KUKA KRL program: EPS_2_25369_MH4A_A_20251215023758.src

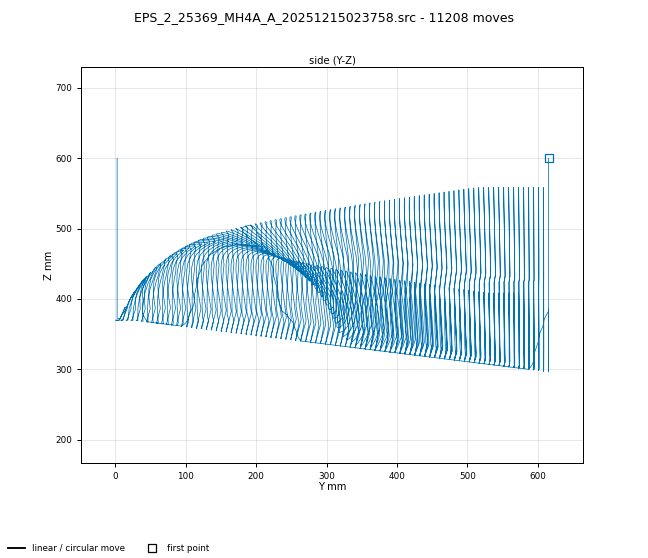
[picture p0: tool path of EPS_2_25369_MH4A_A_20251215023758.src, 11208 of 11210 moves have a stored position in this frame; points joined in program order, loops and branches not executed]
&ACCESS RVP
&REL 4
&COMMENT QRS 19112012
&PARAM EDITMASK = *
DEF PART()
EXT BAS (BAS_COMMAND :IN,REAL :IN )
INT I
BAS (#INITMOV,0 )

;KUKA QRS Post kuka4.cps  Date:22-06-2017 !

File_ID=2957

QRS_PRE_INIT()

;Init var - Until changes are made in qrs_pre_init
Outlet_Square_prg=0
Inlet_1_Square_prg=0
Inlet_2_Square_prg=0
Inlet_3_Square_prg=0
Inlet_4_Square_prg=0
Inlet_5_Square_prg=0

Outlet_1={X 0.000, Y 515.060, Z 433.000, B 0.000, E1 0.000 }
Inlet_1={X 0.000, Y 526.090, Z 283.000, B 0.000, E1 89.000 }
Outlet_1_type=251
Inlet_1_type=251
;QRS#1=Sidecore dimensions
;QRS#2=250-10" PVC SDR 35
;QRS#3=250-10" PVC SDR 35
;QRS#4=
;QRS#5=
;QRS#6=
;QRS#7=
;QRS#8=
;QRS#9=14M PSX
;QRS#10=14M PSX
;QRS#11=
;QRS#12=
;QRS#13=
;QRS#14=
;QRS#15=
;QRS#16=1220x127x838 2,75'
;QRS#17=EPS Height
;QRS#18=558,5
;QRS#19=*
;QRS#20= UPDATED VERSION 22-06-2017
;QRS#21=*
Outlet_Square=0100
Inlet_1_Square=0100
Inlet_2_Square=0
Inlet_3_Square=0
Inlet_4_Square=0
Inlet_5_Square=0
Mill_Square=1
Outlet_Square_Prg=205
Inlet_1_Square_prg=205

QRS_INIT()

$ADVANCE=5

; T1
PTP {E1 173.504,E2 173.504}
PTP {X 0,Y 615.497,A -85,B 0,C 180,E1 173.504,E2 173.504,E3 0,E4 0,E5 0,E6 0}
QRS_SPEED_INIT()
LIN {X 0,Y 615.497,Z 600,A -85,B 0,C 180,E1 173.504,E2 173.504,E3 0,E4 0,E5 0,E6 0} C_VEL
LIN {X 0,Y 615.497,Z 397.017,A -85,B 0,C 180,E1 173.504,E2 173.504} C_VEL
LIN {X 0,Y 615.497,Z 386.319,A -85,B 0,C 180,E1 173.504,E2 173.504} C_VEL
LIN {X 0,Y 615.495,Z 384.629,A -85,B 0,C 180,E1 173.417,E2 173.417} C_VEL
LIN {X 0,Y 615.498,Z 376.216,A -85,B 0,C 180,E1 172.289,E2 172.289} C_VEL
LIN {X 0,Y 615.497,Z 367.233,A -85,B 0,C 180,E1 171.298,E2 171.298} C_VEL
LIN {X 0,Y 615.496,Z 356.352,A -85,B 0,C 180,E1 170.304,E2 170.304} C_VEL
LIN {X 0,Y 615.497,Z 343.901,A -85,B 0,C 180,E1 169.382,E2 169.382} C_VEL
LIN {X 0,Y 615.499,Z 331.514,A -85,B 0,C 180,E1 168.64,E2 168.64} C_VEL
LIN {X 0,Y 615.496,Z 319.313,A -85,B 0,C 180,E1 168.056,E2 168.056} C_VEL
LIN {X 0,Y 615.496,Z 305.868,A -85,B 0,C 180,E1 167.554,E2 167.554} C_VEL
LIN {X 0,Y 615.496,Z 297.285,A -85,B 0,C 180,E1 167.281,E2 167.281} C_VEL
LIN {X 0,Y 615.498,Z 296.435,A -85,B 0,C 180,E1 167.135,E2 167.135} C_VEL
LIN {X 0,Y 615.491,Z 296.315,A -85,B 0,C 180,E1 164.774,E2 164.774} C_VEL
LIN {X 0,Y 615.479,Z 296.31,A -85,B 0,C 180,E1 162.043,E2 162.043} C_VEL
LIN {X 0,Y 615.496,Z 296.324,A -85,B 0,C 180,E1 159.269,E2 159.269} C_VEL
LIN {X 0,Y 615.477,Z 296.311,A -85,B 0,C 180,E1 156.443,E2 156.443} C_VEL
LIN {X 0,Y 615.478,Z 296.31,A -85,B 0,C 180,E1 154.284,E2 154.284} C_VEL
LIN {X 0,Y 615.486,Z 296.32,A -85,B 0,C 180,E1 151.55,E2 151.55} C_VEL
LIN {X 0,Y 615.486,Z 296.314,A -85,B 0,C 180,E1 148.915,E2 148.915} C_VEL
LIN {X 0,Y 615.478,Z 296.31,A -85,B 0,C 180,E1 146.468,E2 146.468} C_VEL
LIN {X 0,Y 615.493,Z 296.308,A -85,B 0,C 180,E1 144.166,E2 144.166} C_VEL
LIN {X 0,Y 615.489,Z 296.313,A -85,B 0,C 180,E1 141.931,E2 141.931} C_VEL
LIN {X 0,Y 615.495,Z 296.322,A -85,B 0,C 180,E1 139.394,E2 139.394} C_VEL
LIN {X 0,Y 615.478,Z 296.31,A -85,B 0,C 180,E1 136.754,E2 136.754} C_VEL
LIN {X 0,Y 615.49,Z 296.314,A -85,B 0,C 180,E1 133.997,E2 133.997} C_VEL
LIN {X 0,Y 615.494,Z 296.32,A -85,B 0,C 180,E1 131.474,E2 131.474} C_VEL
LIN {X 0,Y 615.478,Z 296.311,A -85,B 0,C 180,E1 128.905,E2 128.905} C_VEL
LIN {X 0,Y 615.487,Z 296.309,A -85,B 0,C 180,E1 126.425,E2 126.425} C_VEL
LIN {X 0,Y 615.498,Z 296.318,A -85,B 0,C 180,E1 123.535,E2 123.535} C_VEL
LIN {X 0,Y 615.478,Z 296.31,A -85,B 0,C 180,E1 120.921,E2 120.921} C_VEL
LIN {X 0,Y 615.493,Z 296.309,A -85,B 0,C 180,E1 118.45,E2 118.45} C_VEL
LIN {X 0,Y 615.499,Z 296.315,A -85,B 0,C 180,E1 115.57,E2 115.57} C_VEL
LIN {X 0,Y 615.482,Z 296.309,A -85,B 0,C 180,E1 112.845,E2 112.845} C_VEL
LIN {X 0,Y 615.491,Z 296.324,A -85,B 0,C 180,E1 110.033,E2 110.033} C_VEL
LIN {X 0,Y 615.477,Z 296.311,A -85,B 0,C 180,E1 107.271,E2 107.271} C_VEL
LIN {X 0,Y 615.488,Z 296.312,A -85,B 0,C 180,E1 104.55,E2 104.55} C_VEL
LIN {X 0,Y 615.493,Z 296.319,A -85,B 0,C 180,E1 101.861,E2 101.861} C_VEL
LIN {X 0,Y 615.479,Z 296.309,A -85,B 0,C 180,E1 99.199,E2 99.199} C_VEL
LIN {X 0,Y 615.488,Z 296.315,A -85,B 0,C 180,E1 96.557,E2 96.557} C_VEL
LIN {X 0,Y 615.491,Z 296.318,A -85,B 0,C 180,E1 93.929,E2 93.929} C_VEL
LIN {X 0,Y 615.48,Z 296.309,A -85,B 0,C 180,E1 91.309,E2 91.309} C_VEL
LIN {X 0,Y 615.488,Z 296.314,A -85,B 0,C 180,E1 88.692,E2 88.692} C_VEL
LIN {X 0,Y 615.492,Z 296.318,A -85,B 0,C 180,E1 86.072,E2 86.072} C_VEL
LIN {X 0,Y 615.48,Z 296.309,A -85,B 0,C 180,E1 83.432,E2 83.432} C_VEL
LIN {X 0,Y 615.487,Z 296.315,A -85,B 0,C 180,E1 80.802,E2 80.802} C_VEL
LIN {X 0,Y 615.489,Z 296.317,A -85,B 0,C 180,E1 78.14,E2 78.14} C_VEL
LIN {X 0,Y 615.482,Z 296.309,A -85,B 0,C 180,E1 75.452,E2 75.452} C_VEL
LIN {X 0,Y 615.489,Z 296.32,A -85,B 0,C 180,E1 72.73,E2 72.73} C_VEL
LIN {X 0,Y 615.479,Z 296.313,A -85,B 0,C 180,E1 69.968,E2 69.968} C_VEL
LIN {X 0,Y 615.482,Z 296.309,A -85,B 0,C 180,E1 67.656,E2 67.656} C_VEL
LIN {X 0,Y 615.485,Z 296.316,A -85,B 0,C 180,E1 65.009,E2 65.009} C_VEL
LIN {X 0,Y 615.487,Z 296.322,A -85,B 0,C 180,E1 62.824,E2 62.824} C_VEL
LIN {X 0,Y 615.477,Z 296.315,A -85,B 0,C 180,E1 60.208,E2 60.208} C_VEL
LIN {X 0,Y 615.493,Z 296.307,A -85,B 0,C 180,E1 57.544,E2 57.544} C_VEL
LIN {X 0,Y 615.486,Z 296.315,A -85,B 0,C 180,E1 55.186,E2 55.186} C_VEL
LIN {X 0,Y 615.497,Z 296.323,A -85,B 0,C 180,E1 52.76,E2 52.76} C_VEL
LIN {X 0,Y 615.481,Z 296.309,A -85,B 0,C 180,E1 49.912,E2 49.912} C_VEL
LIN {X 0,Y 615.496,Z 296.307,A -85,B 0,C 180,E1 47.649,E2 47.649} C_VEL
LIN {X 0,Y 615.496,Z 296.326,A -85,B 0,C 180,E1 44.934,E2 44.934} C_VEL
LIN {X 0,Y 615.482,Z 296.309,A -85,B 0,C 180,E1 42.081,E2 42.081} C_VEL
LIN {X 0,Y 615.492,Z 296.308,A -85,B 0,C 180,E1 39.75,E2 39.75} C_VEL
LIN {X 0,Y 615.493,Z 296.322,A -85,B 0,C 180,E1 36.939,E2 36.939} C_VEL
LIN {X 0,Y 615.488,Z 296.307,A -85,B 0,C 180,E1 34.022,E2 34.022} C_VEL
LIN {X 0,Y 615.491,Z 296.325,A -85,B 0,C 180,E1 31.088,E2 31.088} C_VEL
LIN {X 0,Y 615.478,Z 296.311,A -85,B 0,C 180,E1 28.451,E2 28.451} C_VEL
LIN {X 0,Y 615.484,Z 296.314,A -85,B 0,C 180,E1 25.716,E2 25.716} C_VEL
LIN {X 0,Y 615.481,Z 296.316,A -85,B 0,C 180,E1 22.845,E2 22.845} C_VEL
LIN {X 0,Y 615.491,Z 296.308,A -85,B 0,C 180,E1 20.033,E2 20.033} C_VEL
LIN {X 0,Y 615.497,Z 296.322,A -85,B 0,C 180,E1 17.27,E2 17.27} C_VEL
LIN {X 0,Y 615.481,Z 296.309,A -85,B 0,C 180,E1 14.549,E2 14.549} C_VEL
LIN {X 0,Y 615.48,Z 296.316,A -85,B 0,C 180,E1 11.861,E2 11.861} C_VEL
LIN {X 0,Y 615.488,Z 296.318,A -85,B 0,C 180,E1 9.199,E2 9.199} C_VEL
LIN {X 0,Y 615.487,Z 296.307,A -85,B 0,C 180,E1 6.557,E2 6.557} C_VEL
LIN {X 0,Y 615.481,Z 296.317,A -85,B 0,C 180,E1 3.929,E2 3.929} C_VEL
LIN {X 0,Y 615.487,Z 296.318,A -85,B 0,C 180,E1 1.309,E2 1.309} C_VEL
LIN {X 0,Y 615.487,Z 296.307,A -85,B 0,C 180,E1 -1.308,E2 -1.308} C_VEL
LIN {X 0,Y 615.48,Z 296.317,A -85,B 0,C 180,E1 -3.928,E2 -3.928} C_VEL
LIN {X 0,Y 615.485,Z 296.318,A -85,B 0,C 180,E1 -6.585,E2 -6.585} C_VEL
LIN {X 0,Y 615.489,Z 296.307,A -85,B 0,C 180,E1 -9.199,E2 -9.199} C_VEL
LIN {X 0,Y 615.477,Z 296.319,A -85,B 0,C 180,E1 -11.861,E2 -11.861} C_VEL
LIN {X 0,Y 615.481,Z 296.317,A -85,B 0,C 180,E1 -14.549,E2 -14.549} C_VEL
LIN {X 0,Y 615.492,Z 296.307,A -85,B 0,C 180,E1 -17.27,E2 -17.27} C_VEL
LIN {X 0,Y 615.493,Z 296.325,A -85,B 0,C 180,E1 -20.033,E2 -20.033} C_VEL
LIN {X 0,Y 615.481,Z 296.31,A -85,B 0,C 180,E1 -22.845,E2 -22.845} C_VEL
LIN {X 0,Y 615.475,Z 296.317,A -85,B 0,C 180,E1 -25.569,E2 -25.569} C_VEL
LIN {X 0,Y 615.483,Z 296.327,A -85,B 0,C 180,E1 -27.915,E2 -27.915} C_VEL
LIN {X 0,Y 615.488,Z 296.319,A -85,B 0,C 180,E1 -30.16,E2 -30.16} C_VEL
LIN {X 0,Y 615.474,Z 296.314,A -85,B 0,C 180,E1 -32.458,E2 -32.458} C_VEL
LIN {X 0,Y 615.49,Z 296.307,A -85,B 0,C 180,E1 -34.815,E2 -34.815} C_VEL
LIN {X 0,Y 615.48,Z 296.313,A -85,B 0,C 180,E1 -37.243,E2 -37.243} C_VEL
LIN {X 0,Y 615.483,Z 296.318,A -85,B 0,C 180,E1 -40.09,E2 -40.09} C_VEL
LIN {X 0,Y 615.477,Z 296.313,A -85,B 0,C 180,E1 -42.354,E2 -42.354} C_VEL
LIN {X 0,Y 615.48,Z 296.312,A -85,B 0,C 180,E1 -45.069,E2 -45.069} C_VEL
LIN {X 0,Y 615.499,Z 296.325,A -85,B 0,C 180,E1 -47.649,E2 -47.649} C_VEL
LIN {X 0,Y 615.477,Z 296.313,A -85,B 0,C 180,E1 -50.25,E2 -50.25} C_VEL
LIN {X 0,Y 615.49,Z 296.551,A -85,B 0,C 180,E1 -51.725,E2 -51.725} C_VEL
LIN {X 0,Y 615.486,Z 308.417,A -85,B 0,C 180,E1 -54.167,E2 -54.167} C_VEL
LIN {X 0,Y 615.484,Z 321.683,A -85,B 0,C 180,E1 -56.765,E2 -56.765} C_VEL
LIN {X 0,Y 615.497,Z 335.072,A -85,B 0,C 180,E1 -59.462,E2 -59.462} C_VEL
LIN {X 0,Y 615.481,Z 348.459,A -85,B 0,C 180,E1 -62.086,E2 -62.086} C_VEL
LIN {X 0,Y 615.487,Z 362.22,A -85,B 0,C 180,E1 -64.719,E2 -64.719} C_VEL
LIN {X 0,Y 615.498,Z 376.558,A -85,B 0,C 180,E1 -67.407,E2 -67.407} C_VEL
LIN {X 0,Y 615.485,Z 392.386,A -85,B 0,C 180,E1 -70.316,E2 -70.316} C_VEL
LIN {X 0,Y 615.483,Z 407.639,A -85,B 0,C 180,E1 -73.072,E2 -73.072} C_VEL
LIN {X 0,Y 615.486,Z 423.238,A -85,B 0,C 180,E1 -75.836,E2 -75.836} C_VEL
LIN {X 0,Y 615.486,Z 424.86,A -85,B 0,C 180,E1 -75.932,E2 -75.932} C_VEL
LIN {X 0,Y 615.493,Z 439.614,A -85,B 0,C 180,E1 -76.169,E2 -76.169} C_VEL
LIN {X 0,Y 615.483,Z 452.944,A -85,B 0,C 180,E1 -76.505,E2 -76.505} C_VEL
LIN {X 0,Y 615.494,Z 466.162,A -85,B 0,C 180,E1 -76.968,E2 -76.968} C_VEL
LIN {X 0,Y 615.497,Z 479.028,A -85,B 0,C 180,E1 -77.555,E2 -77.555} C_VEL
LIN {X 0,Y 615.498,Z 490.783,A -85,B 0,C 180,E1 -78.224,E2 -78.224} C_VEL
LIN {X 0,Y 615.496,Z 501.416,A -85,B 0,C 180,E1 -78.958,E2 -78.958} C_VEL
LIN {X 0,Y 615.498,Z 511.648,A -85,B 0,C 180,E1 -79.806,E2 -79.806} C_VEL
LIN {X 0,Y 615.498,Z 521.593,A -85,B 0,C 180,E1 -80.802,E2 -80.802} C_VEL
LIN {X 0,Y 615.496,Z 531.077,A -85,B 0,C 180,E1 -81.96,E2 -81.96} C_VEL
LIN {X 0,Y 615.496,Z 538.654,A -85,B 0,C 180,E1 -83.101,E2 -83.101} C_VEL
LIN {X 0,Y 615.499,Z 544.073,A -85,B 0,C 180,E1 -84.102,E2 -84.102} C_VEL
LIN {X 0,Y 615.495,Z 549.685,A -85,B 0,C 180,E1 -85.416,E2 -85.416} C_VEL
LIN {X 0,Y 615.495,Z 553.755,A -85,B 0,C 180,E1 -86.728,E2 -86.728} C_VEL
LIN {X 0,Y 615.499,Z 556.406,A -85,B 0,C 180,E1 -88.038,E2 -88.038} C_VEL
LIN {X 0,Y 615.494,Z 557.723,A -85,B 0,C 180,E1 -89.346,E2 -89.346} C_VEL
LIN {X 0,Y 615.494,Z 557.722,A -85,B 0,C 180,E1 -90.655,E2 -90.655} C_VEL
LIN {X 0,Y 615.499,Z 556.404,A -85,B 0,C 180,E1 -91.964,E2 -91.964} C_VEL
LIN {X 0,Y 615.495,Z 553.752,A -85,B 0,C 180,E1 -93.273,E2 -93.273} C_VEL
LIN {X 0,Y 615.495,Z 549.681,A -85,B 0,C 180,E1 -94.585,E2 -94.585} C_VEL
LIN {X 0,Y 615.499,Z 544.067,A -85,B 0,C 180,E1 -95.899,E2 -95.899} C_VEL
LIN {X 0,Y 615.496,Z 538.65,A -85,B 0,C 180,E1 -96.9,E2 -96.9} C_VEL
LIN {X 0,Y 615.496,Z 531.068,A -85,B 0,C 180,E1 -98.041,E2 -98.041} C_VEL
LIN {X 0,Y 615.498,Z 521.582,A -85,B 0,C 180,E1 -99.199,E2 -99.199} C_VEL
LIN {X 0,Y 615.498,Z 511.636,A -85,B 0,C 180,E1 -100.195,E2 -100.195} C_VEL
LIN {X 0,Y 615.498,Z 500.378,A -85,B 0,C 180,E1 -101.118,E2 -101.118} C_VEL
LIN {X 0,Y 615.498,Z 489.406,A -85,B 0,C 180,E1 -101.861,E2 -101.861} C_VEL
LIN {X 0,Y 615.498,Z 477.317,A -85,B 0,C 180,E1 -102.53,E2 -102.53} C_VEL
LIN {X 0,Y 615.492,Z 463.915,A -85,B 0,C 180,E1 -103.118,E2 -103.118} C_VEL
LIN {X 0,Y 615.484,Z 449.877,A -85,B 0,C 180,E1 -103.58,E2 -103.58} C_VEL
LIN {X 0,Y 615.491,Z 435.698,A -85,B 0,C 180,E1 -103.904,E2 -103.904} C_VEL
LIN {X 0,Y 615.486,Z 424.187,A -85,B 0,C 180,E1 -104.087,E2 -104.087} C_VEL
LIN {X 0,Y 615.487,Z 422.724,A -85,B 0,C 180,E1 -104.241,E2 -104.241} C_VEL
LIN {X 0,Y 615.483,Z 407.632,A -85,B 0,C 180,E1 -106.929,E2 -106.929} C_VEL
LIN {X 0,Y 615.485,Z 392.379,A -85,B 0,C 180,E1 -109.686,E2 -109.686} C_VEL
LIN {X 0,Y 615.498,Z 376.555,A -85,B 0,C 180,E1 -112.594,E2 -112.594} C_VEL
LIN {X 0,Y 615.487,Z 362.216,A -85,B 0,C 180,E1 -115.281,E2 -115.281} C_VEL
LIN {X 0,Y 615.481,Z 348.452,A -85,B 0,C 180,E1 -117.916,E2 -117.916} C_VEL
LIN {X 0,Y 615.497,Z 335.065,A -85,B 0,C 180,E1 -120.539,E2 -120.539} C_VEL
LIN {X 0,Y 615.485,Z 321.676,A -85,B 0,C 180,E1 -123.237,E2 -123.237} C_VEL
LIN {X 0,Y 615.495,Z 304.925,A -85,B 0,C 180,E1 -126.129,E2 -126.129} C_VEL
LIN {X 0,Y 615.499,Z 296.412,A -85,B 0,C 180,E1 -127.65,E2 -127.65} C_VEL
LIN {X 0,Y 615.489,Z 296.314,A -85,B 0,C 180,E1 -130.089,E2 -130.089} C_VEL
LIN {X 0,Y 615.495,Z 296.307,A -85,B 0,C 180,E1 -132.353,E2 -132.353} C_VEL
LIN {X 0,Y 615.482,Z 296.313,A -85,B 0,C 180,E1 -135.069,E2 -135.069} C_VEL
LIN {X 0,Y 615.491,Z 296.315,A -85,B 0,C 180,E1 -137.92,E2 -137.92} C_VEL
LIN {X 0,Y 615.491,Z 296.308,A -85,B 0,C 180,E1 -140.25,E2 -140.25} C_VEL
LIN {X 0,Y 615.488,Z 296.314,A -85,B 0,C 180,E1 -143.064,E2 -143.064} C_VEL
LIN {X 0,Y 615.491,Z 296.311,A -85,B 0,C 180,E1 -145.978,E2 -145.978} C_VEL
LIN {X 0,Y 615.482,Z 296.309,A -85,B 0,C 180,E1 -148.314,E2 -148.314} C_VEL
LIN {X 0,Y 615.479,Z 296.31,A -85,B 0,C 180,E1 -150.593,E2 -150.593} C_VEL
LIN {X 0,Y 615.498,Z 296.312,A -85,B 0,C 180,E1 -152.954,E2 -152.954} C_VEL
LIN {X 0,Y 615.492,Z 296.308,A -85,B 0,C 180,E1 -155.991,E2 -155.991} C_VEL
LIN {X 0,Y 615.479,Z 296.311,A -85,B 0,C 180,E1 -158.568,E2 -158.568} C_VEL
LIN {X 0,Y 615.492,Z 296.321,A -85,B 0,C 180,E1 -161.395,E2 -161.395} C_VEL
LIN {X 0,Y 615.478,Z 296.31,A -85,B 0,C 180,E1 -164.095,E2 -164.095} C_VEL
LIN {X 0,Y 615.498,Z 296.465,A -85,B 0,C 180,E1 -165.24,E2 -165.24} C_VEL
LIN {X 0,Y 615.496,Z 297.227,A -85,B 0,C 180,E1 -165.367,E2 -165.367} C_VEL
LIN {X 0,Y 615.497,Z 314.531,A -85,B 0,C 180,E1 -165.95,E2 -165.95} C_VEL
LIN {X 0,Y 615.496,Z 327.969,A -85,B 0,C 180,E1 -166.547,E2 -166.547} C_VEL
LIN {X 0,Y 615.498,Z 341.296,A -85,B 0,C 180,E1 -167.303,E2 -167.303} C_VEL
LIN {X 0,Y 615.497,Z 353.173,A -85,B 0,C 180,E1 -168.14,E2 -168.14} C_VEL
LIN {X 0,Y 615.496,Z 364.4,A -85,B 0,C 180,E1 -169.109,E2 -169.109} C_VEL
LIN {X 0,Y 615.499,Z 374.182,A -85,B 0,C 180,E1 -170.138,E2 -170.138} C_VEL
LIN {X 0,Y 615.496,Z 383.191,A -85,B 0,C 180,E1 -171.298,E2 -171.298} C_VEL
LIN {X 0,Y 615.496,Z 390.469,A -85,B 0,C 180,E1 -172.455,E2 -172.455} C_VEL
LIN {X 0,Y 615.497,Z 396.954,A -85,B 0,C 180,E1 -173.773,E2 -173.773} C_VEL
LIN {X 0,Y 615.494,Z 401.838,A -85,B 0,C 180,E1 -175.087,E2 -175.087} C_VEL
LIN {X 0,Y 615.493,Z 404.482,A -85,B 0,C 180,E1 -176.072,E2 -176.072} C_VEL
LIN {X 0,Y 615.496,Z 406.836,A -85,B 0,C 180,E1 -177.382,E2 -177.382} C_VEL
LIN {X 0,Y 615.496,Z 407.817,A -85,B 0,C 180,E1 -178.692,E2 -178.692} C_VEL
LIN {X 0,Y 615.493,Z 407.521,A -85,B 0,C 180,E1 -180,E2 -180} C_VEL
LIN {X 0,Y 615.497,Z 405.934,A -85,B 0,C 180,E1 -181.309,E2 -181.309} C_VEL
LIN {X 0,Y 615.494,Z 402.95,A -85,B 0,C 180,E1 -182.618,E2 -182.618} C_VEL
LIN {X 0,Y 615.495,Z 398.558,A -85,B 0,C 180,E1 -183.929,E2 -183.929} C_VEL
LIN {X 0,Y 615.496,Z 394.226,A -85,B 0,C 180,E1 -184.913,E2 -184.913} C_VEL
LIN {X 0,Y 615.498,Z 388.923,A -85,B 0,C 180,E1 -185.899,E2 -185.899} C_VEL
LIN {X 0,Y 615.495,Z 384.629,A -85,B 0,C 180,E1 -186.583,E2 -186.583} C_VEL
LIN {X 0,Y 614.828,Z 381.592,A -85,B 0,C 180,E1 -187.043,E2 -187.043} C_VEL
LIN {X 0,Y 611.986,Z 376.35,A -85,B 0,C 180,E1 -187.78,E2 -187.78} C_VEL
LIN {X 0,Y 609.133,Z 370.491,A -85,B 0,C 180,E1 -188.49,E2 -188.49} C_VEL
LIN {X 0,Y 608.473,Z 366.548,A -85,B 0,C 180,E1 -188.908,E2 -188.908} C_VEL
LIN {X 0,Y 608.497,Z 355.613,A -85,B 0,C 180,E1 -189.893,E2 -189.893} C_VEL
LIN {X 0,Y 608.528,Z 343.269,A -85,B 0,C 180,E1 -190.803,E2 -190.803} C_VEL
LIN {X 0,Y 608.558,Z 331.794,A -85,B 0,C 180,E1 -191.491,E2 -191.491} C_VEL
LIN {X 0,Y 608.575,Z 319.619,A -85,B 0,C 180,E1 -192.082,E2 -192.082} C_VEL
LIN {X 0,Y 608.588,Z 306.233,A -85,B 0,C 180,E1 -192.59,E2 -192.59} C_VEL
LIN {X 0,Y 608.558,Z 297.968,A -85,B 0,C 180,E1 -192.866,E2 -192.866} C_VEL
LIN {X 0,Y 608.495,Z 297.381,A -85,B 0,C 180,E1 -193.016,E2 -193.016} C_VEL
LIN {X 0,Y 608.472,Z 297.313,A -85,B 0,C 180,E1 -195.406,E2 -195.406} C_VEL
LIN {X 0,Y 608.445,Z 297.315,A -85,B 0,C 180,E1 -198.172,E2 -198.172} C_VEL
LIN {X 0,Y 608.46,Z 297.319,A -85,B 0,C 180,E1 -200.982,E2 -200.982} C_VEL
LIN {X 0,Y 608.454,Z 297.317,A -85,B 0,C 180,E1 -203.124,E2 -203.124} C_VEL
LIN {X 0,Y 608.465,Z 297.311,A -85,B 0,C 180,E1 -205.719,E2 -205.719} C_VEL
LIN {X 0,Y 608.451,Z 297.316,A -85,B 0,C 180,E1 -208.267,E2 -208.267} C_VEL
LIN {X 0,Y 608.478,Z 297.318,A -85,B 0,C 180,E1 -210.545,E2 -210.545} C_VEL
LIN {X 0,Y 608.458,Z 297.318,A -85,B 0,C 180,E1 -212.88,E2 -212.88} C_VEL
LIN {X 0,Y 608.445,Z 297.314,A -85,B 0,C 180,E1 -215.278,E2 -215.278} C_VEL
LIN {X 0,Y 608.47,Z 297.311,A -85,B 0,C 180,E1 -217.747,E2 -217.747} C_VEL
LIN {X 0,Y 608.458,Z 297.319,A -85,B 0,C 180,E1 -220.329,E2 -220.329} C_VEL
LIN {X 0,Y 608.45,Z 297.315,A -85,B 0,C 180,E1 -222.961,E2 -222.961} C_VEL
LIN {X 0,Y 608.462,Z 297.312,A -85,B 0,C 180,E1 -225.736,E2 -225.736} C_VEL
LIN {X 0,Y 608.466,Z 297.316,A -85,B 0,C 180,E1 -228.658,E2 -228.658} C_VEL
LIN {X 0,Y 608.469,Z 297.312,A -85,B 0,C 180,E1 -231.76,E2 -231.76} C_VEL
LIN {X 0,Y 608.453,Z 297.317,A -85,B 0,C 180,E1 -233.954,E2 -233.954} C_VEL
LIN {X 0,Y 608.472,Z 297.319,A -85,B 0,C 180,E1 -236.329,E2 -236.329} C_VEL
LIN {X 0,Y 608.45,Z 297.315,A -85,B 0,C 180,E1 -238.733,E2 -238.733} C_VEL
LIN {X 0,Y 608.475,Z 297.31,A -85,B 0,C 180,E1 -241.381,E2 -241.381} C_VEL
LIN {X 0,Y 608.483,Z 297.317,A -85,B 0,C 180,E1 -244.278,E2 -244.278} C_VEL
LIN {X 0,Y 608.45,Z 297.313,A -85,B 0,C 180,E1 -246.876,E2 -246.876} C_VEL
LIN {X 0,Y 608.467,Z 297.316,A -85,B 0,C 180,E1 -249.726,E2 -249.726} C_VEL
LIN {X 0,Y 608.451,Z 297.315,A -85,B 0,C 180,E1 -252.523,E2 -252.523} C_VEL
LIN {X 0,Y 608.475,Z 297.311,A -85,B 0,C 180,E1 -255.279,E2 -255.279} C_VEL
LIN {X 0,Y 608.468,Z 297.32,A -85,B 0,C 180,E1 -258,E2 -258} C_VEL
LIN {X 0,Y 608.467,Z 297.311,A -85,B 0,C 180,E1 -260.694,E2 -260.694} C_VEL
LIN {X 0,Y 608.465,Z 297.314,A -85,B 0,C 180,E1 -263.384,E2 -263.384} C_VEL
LIN {X 0,Y 608.46,Z 297.318,A -85,B 0,C 180,E1 -266.025,E2 -266.025} C_VEL
LIN {X 0,Y 608.466,Z 297.311,A -85,B 0,C 180,E1 -268.676,E2 -268.676} C_VEL
LIN {X 0,Y 608.472,Z 297.314,A -85,B 0,C 180,E1 -271.323,E2 -271.323} C_VEL
LIN {X 0,Y 608.459,Z 297.317,A -85,B 0,C 180,E1 -273.973,E2 -273.973} C_VEL
LIN {X 0,Y 608.465,Z 297.311,A -85,B 0,C 180,E1 -276.632,E2 -276.632} C_VEL
LIN {X 0,Y 608.473,Z 297.315,A -85,B 0,C 180,E1 -279.305,E2 -279.305} C_VEL
LIN {X 0,Y 608.464,Z 297.314,A -85,B 0,C 180,E1 -281.999,E2 -281.999} C_VEL
LIN {X 0,Y 608.473,Z 297.31,A -85,B 0,C 180,E1 -284.72,E2 -284.72} C_VEL
LIN {X 0,Y 608.454,Z 297.323,A -85,B 0,C 180,E1 -287.476,E2 -287.476} C_VEL
LIN {X 0,Y 608.459,Z 297.312,A -85,B 0,C 180,E1 -290.273,E2 -290.273} C_VEL
LIN {X 0,Y 608.461,Z 297.311,A -85,B 0,C 180,E1 -292.475,E2 -292.475} C_VEL
LIN {X 0,Y 608.457,Z 297.322,A -85,B 0,C 180,E1 -295.3,E2 -295.3} C_VEL
LIN {X 0,Y 608.448,Z 297.32,A -85,B 0,C 180,E1 -297.517,E2 -297.517} C_VEL
LIN {X 0,Y 608.459,Z 297.313,A -85,B 0,C 180,E1 -299.969,E2 -299.969} C_VEL
LIN {X 0,Y 608.467,Z 297.311,A -85,B 0,C 180,E1 -302.522,E2 -302.522} C_VEL
LIN {X 0,Y 608.444,Z 297.323,A -85,B 0,C 180,E1 -305.277,E2 -305.277} C_VEL
LIN {X 0,Y 608.468,Z 297.312,A -85,B 0,C 180,E1 -307.745,E2 -307.745} C_VEL
LIN {X 0,Y 608.45,Z 297.313,A -85,B 0,C 180,E1 -310.328,E2 -310.328} C_VEL
LIN {X 0,Y 608.484,Z 297.315,A -85,B 0,C 180,E1 -313.31,E2 -313.31} C_VEL
LIN {X 0,Y 608.468,Z 297.31,A -85,B 0,C 180,E1 -316.13,E2 -316.13} C_VEL
LIN {X 0,Y 608.46,Z 297.319,A -85,B 0,C 180,E1 -318.823,E2 -318.823} C_VEL
LIN {X 0,Y 608.473,Z 297.313,A -85,B 0,C 180,E1 -321.412,E2 -321.412} C_VEL
LIN {X 0,Y 608.476,Z 297.309,A -85,B 0,C 180,E1 -323.949,E2 -323.949} C_VEL
LIN {X 0,Y 608.463,Z 297.313,A -85,B 0,C 180,E1 -326.329,E2 -326.329} C_VEL
LIN {X 0,Y 608.476,Z 297.318,A -85,B 0,C 180,E1 -328.726,E2 -328.726} C_VEL
LIN {X 0,Y 608.466,Z 297.313,A -85,B 0,C 180,E1 -331.379,E2 -331.379} C_VEL
LIN {X 0,Y 608.441,Z 297.314,A -85,B 0,C 180,E1 -333.964,E2 -333.964} C_VEL
LIN {X 0,Y 608.468,Z 297.312,A -85,B 0,C 180,E1 -336.155,E2 -336.155} C_VEL
LIN {X 0,Y 608.452,Z 297.318,A -85,B 0,C 180,E1 -339.018,E2 -339.018} C_VEL
LIN {X 0,Y 608.446,Z 297.313,A -85,B 0,C 180,E1 -341.828,E2 -341.828} C_VEL
LIN {X 0,Y 608.473,Z 297.32,A -85,B 0,C 180,E1 -344.594,E2 -344.594} C_VEL
LIN {X 0,Y 608.475,Z 297.31,A -85,B 0,C 180,E1 -347.323,E2 -347.323} C_VEL
LIN {X 0,Y 608.454,Z 297.315,A -85,B 0,C 180,E1 -350.022,E2 -350.022} C_VEL
LIN {X 0,Y 608.479,Z 297.316,A -85,B 0,C 180,E1 -352.701,E2 -352.701} C_VEL
LIN {X 0,Y 608.454,Z 297.312,A -85,B 0,C 180,E1 -355.362,E2 -355.362} C_VEL
LIN {X 0,Y 608.453,Z 297.316,A -85,B 0,C 180,E1 -358.014,E2 -358.014} C_VEL
LIN {X 0,Y 608.478,Z 297.315,A -85,B 0,C 180,E1 -360.662,E2 -360.662} C_VEL
LIN {X 0,Y 608.476,Z 297.309,A -85,B 0,C 180,E1 -363.311,E2 -363.311} C_VEL
LIN {X 0,Y 608.452,Z 297.317,A -85,B 0,C 180,E1 -365.967,E2 -365.967} C_VEL
LIN {X 0,Y 608.454,Z 297.316,A -85,B 0,C 180,E1 -368.636,E2 -368.636} C_VEL
LIN {X 0,Y 608.473,Z 297.31,A -85,B 0,C 180,E1 -371.324,E2 -371.324} C_VEL
LIN {X 0,Y 608.461,Z 297.32,A -85,B 0,C 180,E1 -374.038,E2 -374.038} C_VEL
LIN {X 0,Y 608.47,Z 297.311,A -85,B 0,C 180,E1 -376.783,E2 -376.783} C_VEL
LIN {X 0,Y 608.455,Z 297.315,A -85,B 0,C 180,E1 -379.57,E2 -379.57} C_VEL
LIN {X 0,Y 608.45,Z 297.316,A -85,B 0,C 180,E1 -382.477,E2 -382.477} C_VEL
LIN {X 0,Y 608.453,Z 297.314,A -85,B 0,C 180,E1 -384.571,E2 -384.571} C_VEL
LIN {X 0,Y 608.482,Z 297.309,A -85,B 0,C 180,E1 -387.21,E2 -387.21} C_VEL
LIN {X 0,Y 608.467,Z 297.321,A -85,B 0,C 180,E1 -389.973,E2 -389.973} C_VEL
LIN {X 0,Y 608.45,Z 297.314,A -85,B 0,C 180,E1 -392.522,E2 -392.522} C_VEL
LIN {X 0,Y 608.442,Z 297.316,A -85,B 0,C 180,E1 -395.278,E2 -395.278} C_VEL
LIN {X 0,Y 608.467,Z 297.32,A -85,B 0,C 180,E1 -397.746,E2 -397.746} C_VEL
LIN {X 0,Y 608.448,Z 297.315,A -85,B 0,C 180,E1 -400.33,E2 -400.33} C_VEL
LIN {X 0,Y 608.449,Z 297.314,A -85,B 0,C 180,E1 -402.96,E2 -402.96} C_VEL
LIN {X 0,Y 608.458,Z 297.322,A -85,B 0,C 180,E1 -405.736,E2 -405.736} C_VEL
LIN {X 0,Y 608.461,Z 297.312,A -85,B 0,C 180,E1 -408.658,E2 -408.658} C_VEL
LIN {X 0,Y 608.494,Z 297.418,A -85,B 0,C 180,E1 -411.471,E2 -411.471} C_VEL
LIN {X 0,Y 608.624,Z 303.732,A -85,B 0,C 180,E1 -412.823,E2 -412.823} C_VEL
LIN {X 0,Y 608.595,Z 317.198,A -85,B 0,C 180,E1 -415.54,E2 -415.54} C_VEL
LIN {X 0,Y 608.632,Z 331.247,A -85,B 0,C 180,E1 -418.306,E2 -418.306} C_VEL
LIN {X 0,Y 608.59,Z 344.634,A -85,B 0,C 180,E1 -420.987,E2 -420.987} C_VEL
LIN {X 0,Y 608.562,Z 358.022,A -85,B 0,C 180,E1 -423.602,E2 -423.602} C_VEL
LIN {X 0,Y 608.526,Z 371.409,A -85,B 0,C 180,E1 -426.158,E2 -426.158} C_VEL
LIN {X 0,Y 608.507,Z 384.796,A -85,B 0,C 180,E1 -428.666,E2 -428.666} C_VEL
LIN {X 0,Y 608.495,Z 400.494,A -85,B 0,C 180,E1 -431.554,E2 -431.554} C_VEL
LIN {X 0,Y 608.463,Z 415.396,A -85,B 0,C 180,E1 -434.251,E2 -434.251} C_VEL
LIN {X 0,Y 608.513,Z 423.943,A -85,B 0,C 180,E1 -435.734,E2 -435.734} C_VEL
LIN {X 0,Y 608.601,Z 427.881,A -85,B 0,C 180,E1 -435.813,E2 -435.813} C_VEL
LIN {X 0,Y 608.59,Z 442.101,A -85,B 0,C 180,E1 -436.066,E2 -436.066} C_VEL
LIN {X 0,Y 608.573,Z 455.575,A -85,B 0,C 180,E1 -436.434,E2 -436.434} C_VEL
LIN {X 0,Y 608.574,Z 468.173,A -85,B 0,C 180,E1 -436.902,E2 -436.902} C_VEL
LIN {X 0,Y 608.539,Z 480.654,A -85,B 0,C 180,E1 -437.495,E2 -437.495} C_VEL
LIN {X 0,Y 608.531,Z 493.435,A -85,B 0,C 180,E1 -438.256,E2 -438.256} C_VEL
LIN {X 0,Y 608.499,Z 504.702,A -85,B 0,C 180,E1 -439.079,E2 -439.079} C_VEL
LIN {X 0,Y 608.473,Z 515.398,A -85,B 0,C 180,E1 -440.024,E2 -440.024} C_VEL
LIN {X 0,Y 608.473,Z 524.829,A -85,B 0,C 180,E1 -441.03,E2 -441.03} C_VEL
LIN {X 0,Y 608.453,Z 533.802,A -85,B 0,C 180,E1 -442.2,E2 -442.2} C_VEL
LIN {X 0,Y 608.441,Z 541.23,A -85,B 0,C 180,E1 -443.4,E2 -443.4} C_VEL
LIN {X 0,Y 608.44,Z 547.57,A -85,B 0,C 180,E1 -444.699,E2 -444.699} C_VEL
LIN {X 0,Y 608.431,Z 552.443,A -85,B 0,C 180,E1 -446.027,E2 -446.027} C_VEL
LIN {X 0,Y 608.424,Z 555.832,A -85,B 0,C 180,E1 -447.352,E2 -447.352} C_VEL
LIN {X 0,Y 608.442,Z 557.831,A -85,B 0,C 180,E1 -448.677,E2 -448.677} C_VEL
LIN {X 0,Y 608.433,Z 558.5,A -85,B 0,C 180,E1 -450.001,E2 -450.001} C_VEL
LIN {X 0,Y 608.442,Z 557.83,A -85,B 0,C 180,E1 -451.324,E2 -451.324} C_VEL
LIN {X 0,Y 608.424,Z 555.83,A -85,B 0,C 180,E1 -452.649,E2 -452.649} C_VEL
LIN {X 0,Y 608.432,Z 552.439,A -85,B 0,C 180,E1 -453.975,E2 -453.975} C_VEL
LIN {X 0,Y 608.44,Z 547.565,A -85,B 0,C 180,E1 -455.303,E2 -455.303} C_VEL
LIN {X 0,Y 608.446,Z 541.208,A -85,B 0,C 180,E1 -456.604,E2 -456.604} C_VEL
LIN {X 0,Y 608.453,Z 533.794,A -85,B 0,C 180,E1 -457.801,E2 -457.801} C_VEL
LIN {X 0,Y 608.473,Z 524.818,A -85,B 0,C 180,E1 -458.971,E2 -458.971} C_VEL
LIN {X 0,Y 608.473,Z 515.385,A -85,B 0,C 180,E1 -459.978,E2 -459.978} C_VEL
LIN {X 0,Y 608.506,Z 504.043,A -85,B 0,C 180,E1 -460.973,E2 -460.973} C_VEL
LIN {X 0,Y 608.535,Z 492.139,A -85,B 0,C 180,E1 -461.83,E2 -461.83} C_VEL
LIN {X 0,Y 608.536,Z 479.062,A -85,B 0,C 180,E1 -462.591,E2 -462.591} C_VEL
LIN {X 0,Y 608.557,Z 466.158,A -85,B 0,C 180,E1 -463.185,E2 -463.185} C_VEL
LIN {X 0,Y 608.587,Z 452.161,A -85,B 0,C 180,E1 -463.673,E2 -463.673} C_VEL
LIN {X 0,Y 608.599,Z 438.422,A -85,B 0,C 180,E1 -464.014,E2 -464.014} C_VEL
LIN {X 0,Y 608.508,Z 424.029,A -85,B 0,C 180,E1 -464.261,E2 -464.261} C_VEL
LIN {X 0,Y 608.468,Z 423.052,A -85,B 0,C 180,E1 -464.379,E2 -464.379} C_VEL
LIN {X 0,Y 608.471,Z 407.739,A -85,B 0,C 180,E1 -467.13,E2 -467.13} C_VEL
LIN {X 0,Y 608.5,Z 394.352,A -85,B 0,C 180,E1 -469.569,E2 -469.569} C_VEL
LIN {X 0,Y 608.531,Z 378.578,A -85,B 0,C 180,E1 -472.492,E2 -472.492} C_VEL
LIN {X 0,Y 608.562,Z 363.752,A -85,B 0,C 180,E1 -475.297,E2 -475.297} C_VEL
LIN {X 0,Y 608.566,Z 348.452,A -85,B 0,C 180,E1 -478.261,E2 -478.261} C_VEL
LIN {X 0,Y 608.606,Z 335.102,A -85,B 0,C 180,E1 -480.915,E2 -480.915} C_VEL
LIN {X 0,Y 608.612,Z 326.996,A -85,B 0,C 180,E1 -482.544,E2 -482.544} C_VEL
LIN {X 0,Y 608.516,Z 307.823,A -85,B 0,C 180,E1 -485.855,E2 -485.855} C_VEL
LIN {X 0,Y 608.484,Z 297.426,A -85,B 0,C 180,E1 -487.725,E2 -487.725} C_VEL
LIN {X 0,Y 608.451,Z 297.314,A -85,B 0,C 180,E1 -490.329,E2 -490.329} C_VEL
LIN {X 0,Y 608.483,Z 297.314,A -85,B 0,C 180,E1 -493.31,E2 -493.31} C_VEL
LIN {X 0,Y 608.474,Z 297.312,A -85,B 0,C 180,E1 -496.131,E2 -496.131} C_VEL
LIN {X 0,Y 608.451,Z 297.313,A -85,B 0,C 180,E1 -498.823,E2 -498.823} C_VEL
LIN {X 0,Y 608.474,Z 297.319,A -85,B 0,C 180,E1 -501.412,E2 -501.412} C_VEL
LIN {X 0,Y 608.482,Z 297.312,A -85,B 0,C 180,E1 -503.95,E2 -503.95} C_VEL
LIN {X 0,Y 608.449,Z 297.313,A -85,B 0,C 180,E1 -506.328,E2 -506.328} C_VEL
LIN {X 0,Y 608.449,Z 297.314,A -85,B 0,C 180,E1 -508.733,E2 -508.733} C_VEL
LIN {X 0,Y 608.478,Z 297.32,A -85,B 0,C 180,E1 -511.38,E2 -511.38} C_VEL
LIN {X 0,Y 608.442,Z 297.315,A -85,B 0,C 180,E1 -513.964,E2 -513.964} C_VEL
LIN {X 0,Y 608.467,Z 297.311,A -85,B 0,C 180,E1 -516.155,E2 -516.155} C_VEL
LIN {X 0,Y 608.468,Z 297.311,A -85,B 0,C 180,E1 -518.309,E2 -518.309} C_VEL
LIN {X 0,Y 608.476,Z 297.32,A -85,B 0,C 180,E1 -521.283,E2 -521.283} C_VEL
LIN {X 0,Y 608.459,Z 297.313,A -85,B 0,C 180,E1 -523.906,E2 -523.906} C_VEL
LIN {X 0,Y 608.508,Z 297.506,A -85,B 0,C 180,E1 -525.152,E2 -525.152} C_VEL
LIN {X 0,Y 608.605,Z 298.578,A -85,B 0,C 180,E1 -525.261,E2 -525.261} C_VEL
LIN {X 0,Y 608.588,Z 313.911,A -85,B 0,C 180,E1 -525.774,E2 -525.774} C_VEL
LIN {X 0,Y 608.563,Z 326.104,A -85,B 0,C 180,E1 -526.306,E2 -526.306} C_VEL
LIN {X 0,Y 608.533,Z 338.504,A -85,B 0,C 180,E1 -526.985,E2 -526.985} C_VEL
LIN {X 0,Y 608.502,Z 350.961,A -85,B 0,C 180,E1 -527.832,E2 -527.832} C_VEL
LIN {X 0,Y 608.491,Z 361.228,A -85,B 0,C 180,E1 -528.677,E2 -528.677} C_VEL
LIN {X 0,Y 608.479,Z 371.374,A -85,B 0,C 180,E1 -529.687,E2 -529.687} C_VEL
LIN {X 0,Y 608.451,Z 379.795,A -85,B 0,C 180,E1 -530.694,E2 -530.694} C_VEL
LIN {X 0,Y 608.462,Z 387.874,A -85,B 0,C 180,E1 -531.866,E2 -531.866} C_VEL
LIN {X 0,Y 608.441,Z 394.324,A -85,B 0,C 180,E1 -533.034,E2 -533.034} C_VEL
LIN {X 0,Y 608.429,Z 400.057,A -85,B 0,C 180,E1 -534.366,E2 -534.366} C_VEL
LIN {X 0,Y 608.431,Z 403.309,A -85,B 0,C 180,E1 -535.362,E2 -535.362} C_VEL
LIN {X 0,Y 608.422,Z 406.394,A -85,B 0,C 180,E1 -536.689,E2 -536.689} C_VEL
LIN {X 0,Y 608.442,Z 408.088,A -85,B 0,C 180,E1 -538.014,E2 -538.014} C_VEL
LIN {X 0,Y 608.437,Z 408.443,A -85,B 0,C 180,E1 -539.338,E2 -539.338} C_VEL
LIN {X 0,Y 608.437,Z 407.507,A -85,B 0,C 180,E1 -540.662,E2 -540.662} C_VEL
LIN {X 0,Y 608.441,Z 405.212,A -85,B 0,C 180,E1 -541.986,E2 -541.986} C_VEL
LIN {X 0,Y 608.427,Z 401.504,A -85,B 0,C 180,E1 -543.311,E2 -543.311} C_VEL
LIN {X 0,Y 608.446,Z 396.323,A -85,B 0,C 180,E1 -544.638,E2 -544.638} C_VEL
LIN {X 0,Y 608.448,Z 391.306,A -85,B 0,C 180,E1 -545.635,E2 -545.635} C_VEL
LIN {X 0,Y 608.461,Z 384.126,A -85,B 0,C 180,E1 -546.8,E2 -546.8} C_VEL
LIN {X 0,Y 608.459,Z 375.205,A -85,B 0,C 180,E1 -547.967,E2 -547.967} C_VEL
LIN {X 0,Y 608.473,Z 366.548,A -85,B 0,C 180,E1 -548.908,E2 -548.908} C_VEL
LIN {X 0,Y 607.807,Z 362.526,A -85,B 0,C 180,E1 -549.311,E2 -549.311} C_VEL
LIN {X 0,Y 604.96,Z 355.809,A -85,B 0,C 180,E1 -549.947,E2 -549.947} C_VEL
LIN {X 0,Y 602.151,Z 348.725,A -85,B 0,C 180,E1 -550.546,E2 -550.546} C_VEL
LIN {X 0,Y 601.543,Z 344.042,A -85,B 0,C 180,E1 -550.888,E2 -550.888} C_VEL
LIN {X 0,Y 601.583,Z 332.008,A -85,B 0,C 180,E1 -551.626,E2 -551.626} C_VEL
LIN {X 0,Y 601.637,Z 319.895,A -85,B 0,C 180,E1 -552.224,E2 -552.224} C_VEL
LIN {X 0,Y 601.68,Z 305.309,A -85,B 0,C 180,E1 -552.78,E2 -552.78} C_VEL
LIN {X 0,Y 601.626,Z 299.231,A -85,B 0,C 180,E1 -552.974,E2 -552.974} C_VEL
LIN {X 0,Y 601.484,Z 298.348,A -85,B 0,C 180,E1 -553.085,E2 -553.085} C_VEL
LIN {X 0,Y 601.415,Z 298.191,A -85,B 0,C 180,E1 -555.592,E2 -555.592} C_VEL
LIN {X 0,Y 601.398,Z 298.192,A -85,B 0,C 180,E1 -557.689,E2 -557.689} C_VEL
LIN {X 0,Y 601.435,Z 298.193,A -85,B 0,C 180,E1 -560.522,E2 -560.522} C_VEL
LIN {X 0,Y 601.422,Z 298.19,A -85,B 0,C 180,E1 -563.411,E2 -563.411} C_VEL
LIN {X 0,Y 601.406,Z 298.195,A -85,B 0,C 180,E1 -566.364,E2 -566.364} C_VEL
LIN {X 0,Y 601.441,Z 298.194,A -85,B 0,C 180,E1 -568.789,E2 -568.789} C_VEL
LIN {X 0,Y 601.423,Z 298.188,A -85,B 0,C 180,E1 -571.455,E2 -571.455} C_VEL
LIN {X 0,Y 601.436,Z 298.189,A -85,B 0,C 180,E1 -574.118,E2 -574.118} C_VEL
LIN {X 0,Y 601.417,Z 298.199,A -85,B 0,C 180,E1 -576.582,E2 -576.582} C_VEL
LIN {X 0,Y 601.418,Z 298.19,A -85,B 0,C 180,E1 -579.126,E2 -579.126} C_VEL
LIN {X 0,Y 601.426,Z 298.189,A -85,B 0,C 180,E1 -581.765,E2 -581.765} C_VEL
LIN {X 0,Y 601.43,Z 298.196,A -85,B 0,C 180,E1 -584.535,E2 -584.535} C_VEL
LIN {X 0,Y 601.417,Z 298.189,A -85,B 0,C 180,E1 -587.33,E2 -587.33} C_VEL
LIN {X 0,Y 601.408,Z 298.195,A -85,B 0,C 180,E1 -590.004,E2 -590.004} C_VEL
LIN {X 0,Y 601.44,Z 298.191,A -85,B 0,C 180,E1 -592.618,E2 -592.618} C_VEL
LIN {X 0,Y 601.409,Z 298.19,A -85,B 0,C 180,E1 -595.067,E2 -595.067} C_VEL
LIN {X 0,Y 601.438,Z 298.187,A -85,B 0,C 180,E1 -597.484,E2 -597.484} C_VEL
LIN {X 0,Y 601.435,Z 298.191,A -85,B 0,C 180,E1 -599.851,E2 -599.851} C_VEL
LIN {X 0,Y 601.414,Z 298.192,A -85,B 0,C 180,E1 -602.639,E2 -602.639} C_VEL
LIN {X 0,Y 601.404,Z 298.19,A -85,B 0,C 180,E1 -605.121,E2 -605.121} C_VEL
LIN {X 0,Y 601.422,Z 298.189,A -85,B 0,C 180,E1 -607.394,E2 -607.394} C_VEL
LIN {X 0,Y 601.408,Z 298.198,A -85,B 0,C 180,E1 -610.19,E2 -610.19} C_VEL
LIN {X 0,Y 601.436,Z 298.186,A -85,B 0,C 180,E1 -613.014,E2 -613.014} C_VEL
LIN {X 0,Y 601.428,Z 298.197,A -85,B 0,C 180,E1 -615.908,E2 -615.908} C_VEL
LIN {X 0,Y 601.419,Z 298.19,A -85,B 0,C 180,E1 -618.541,E2 -618.541} C_VEL
LIN {X 0,Y 601.418,Z 298.19,A -85,B 0,C 180,E1 -621.262,E2 -621.262} C_VEL
LIN {X 0,Y 601.442,Z 298.194,A -85,B 0,C 180,E1 -623.963,E2 -623.963} C_VEL
LIN {X 0,Y 601.427,Z 298.188,A -85,B 0,C 180,E1 -626.65,E2 -626.65} C_VEL
LIN {X 0,Y 601.453,Z 298.188,A -85,B 0,C 180,E1 -629.33,E2 -629.33} C_VEL
LIN {X 0,Y 601.438,Z 298.192,A -85,B 0,C 180,E1 -632.008,E2 -632.008} C_VEL
LIN {X 0,Y 601.417,Z 298.189,A -85,B 0,C 180,E1 -634.691,E2 -634.691} C_VEL
LIN {X 0,Y 601.444,Z 298.192,A -85,B 0,C 180,E1 -637.384,E2 -637.384} C_VEL
LIN {X 0,Y 601.44,Z 298.189,A -85,B 0,C 180,E1 -640.094,E2 -640.094} C_VEL
LIN {X 0,Y 601.42,Z 298.189,A -85,B 0,C 180,E1 -642.827,E2 -642.827} C_VEL
LIN {X 0,Y 601.416,Z 298.198,A -85,B 0,C 180,E1 -645.59,E2 -645.59} C_VEL
LIN {X 0,Y 601.422,Z 298.188,A -85,B 0,C 180,E1 -648.391,E2 -648.391} C_VEL
LIN {X 0,Y 601.412,Z 298.197,A -85,B 0,C 180,E1 -651.238,E2 -651.238} C_VEL
LIN {X 0,Y 601.452,Z 298.185,A -85,B 0,C 180,E1 -654.14,E2 -654.14} C_VEL
LIN {X 0,Y 601.452,Z 298.191,A -85,B 0,C 180,E1 -657.11,E2 -657.11} C_VEL
LIN {X 0,Y 601.419,Z 298.198,A -85,B 0,C 180,E1 -659.392,E2 -659.392} C_VEL
LIN {X 0,Y 601.415,Z 298.192,A -85,B 0,C 180,E1 -661.725,E2 -661.725} C_VEL
LIN {X 0,Y 601.429,Z 298.187,A -85,B 0,C 180,E1 -664.117,E2 -664.117} C_VEL
LIN {X 0,Y 601.437,Z 298.193,A -85,B 0,C 180,E1 -667.382,E2 -667.382} C_VEL
LIN {X 0,Y 601.409,Z 298.19,A -85,B 0,C 180,E1 -669.994,E2 -669.994} C_VEL
LIN {X 0,Y 601.415,Z 298.193,A -85,B 0,C 180,E1 -672.669,E2 -672.669} C_VEL
LIN {X 0,Y 601.423,Z 298.192,A -85,B 0,C 180,E1 -675.481,E2 -675.481} C_VEL
LIN {X 0,Y 601.424,Z 298.19,A -85,B 0,C 180,E1 -678.406,E2 -678.406} C_VEL
LIN {X 0,Y 601.438,Z 298.195,A -85,B 0,C 180,E1 -680.875,E2 -680.875} C_VEL
LIN {X 0,Y 601.442,Z 298.186,A -85,B 0,C 180,E1 -683.733,E2 -683.733} C_VEL
LIN {X 0,Y 601.43,Z 298.187,A -85,B 0,C 180,E1 -686.063,E2 -686.063} C_VEL
LIN {X 0,Y 601.43,Z 298.194,A -85,B 0,C 180,E1 -689.058,E2 -689.058} C_VEL
LIN {X 0,Y 601.426,Z 298.19,A -85,B 0,C 180,E1 -691.373,E2 -691.373} C_VEL
LIN {X 0,Y 601.401,Z 298.191,A -85,B 0,C 180,E1 -693.636,E2 -693.636} C_VEL
LIN {X 0,Y 601.418,Z 298.197,A -85,B 0,C 180,E1 -696.589,E2 -696.589} C_VEL
LIN {X 0,Y 601.425,Z 298.188,A -85,B 0,C 180,E1 -699.478,E2 -699.478} C_VEL
LIN {X 0,Y 601.4,Z 298.196,A -85,B 0,C 180,E1 -702.312,E2 -702.312} C_VEL
LIN {X 0,Y 601.416,Z 298.196,A -85,B 0,C 180,E1 -704.409,E2 -704.409} C_VEL
LIN {X 0,Y 601.421,Z 298.19,A -85,B 0,C 180,E1 -707.172,E2 -707.172} C_VEL
LIN {X 0,Y 601.431,Z 298.189,A -85,B 0,C 180,E1 -709.905,E2 -709.905} C_VEL
LIN {X 0,Y 601.448,Z 298.193,A -85,B 0,C 180,E1 -712.615,E2 -712.615} C_VEL
LIN {X 0,Y 601.423,Z 298.188,A -85,B 0,C 180,E1 -715.308,E2 -715.308} C_VEL
LIN {X 0,Y 601.423,Z 298.192,A -85,B 0,C 180,E1 -717.991,E2 -717.991} C_VEL
LIN {X 0,Y 601.449,Z 298.19,A -85,B 0,C 180,E1 -720.669,E2 -720.669} C_VEL
LIN {X 0,Y 601.427,Z 298.187,A -85,B 0,C 180,E1 -723.349,E2 -723.349} C_VEL
LIN {X 0,Y 601.406,Z 298.196,A -85,B 0,C 180,E1 -726.037,E2 -726.037} C_VEL
LIN {X 0,Y 601.434,Z 298.19,A -85,B 0,C 180,E1 -728.738,E2 -728.738} C_VEL
LIN {X 0,Y 601.429,Z 298.188,A -85,B 0,C 180,E1 -731.458,E2 -731.458} C_VEL
LIN {X 0,Y 601.412,Z 298.2,A -85,B 0,C 180,E1 -734.206,E2 -734.206} C_VEL
LIN {X 0,Y 601.428,Z 298.188,A -85,B 0,C 180,E1 -736.986,E2 -736.986} C_VEL
LIN {X 0,Y 601.407,Z 298.196,A -85,B 0,C 180,E1 -739.809,E2 -739.809} C_VEL
LIN {X 0,Y 601.404,Z 298.192,A -85,B 0,C 180,E1 -742.683,E2 -742.683} C_VEL
LIN {X 0,Y 601.401,Z 298.191,A -85,B 0,C 180,E1 -744.879,E2 -744.879} C_VEL
LIN {X 0,Y 601.417,Z 298.198,A -85,B 0,C 180,E1 -747.867,E2 -747.867} C_VEL
LIN {X 0,Y 601.442,Z 298.192,A -85,B 0,C 180,E1 -750.163,E2 -750.163} C_VEL
LIN {X 0,Y 601.413,Z 298.19,A -85,B 0,C 180,E1 -752.716,E2 -752.716} C_VEL
LIN {X 0,Y 601.411,Z 298.19,A -85,B 0,C 180,E1 -755.116,E2 -755.116} C_VEL
LIN {X 0,Y 601.43,Z 298.191,A -85,B 0,C 180,E1 -757.419,E2 -757.419} C_VEL
LIN {X 0,Y 601.407,Z 298.197,A -85,B 0,C 180,E1 -759.995,E2 -759.995} C_VEL
LIN {X 0,Y 601.406,Z 298.191,A -85,B 0,C 180,E1 -762.671,E2 -762.671} C_VEL
LIN {X 0,Y 601.42,Z 298.196,A -85,B 0,C 180,E1 -765.483,E2 -765.483} C_VEL
LIN {X 0,Y 601.422,Z 298.19,A -85,B 0,C 180,E1 -768.407,E2 -768.407} C_VEL
LIN {X 0,Y 601.456,Z 298.322,A -85,B 0,C 180,E1 -771.229,E2 -771.229} C_VEL
LIN {X 0,Y 601.811,Z 302.672,A -85,B 0,C 180,E1 -772.188,E2 -772.188} C_VEL
LIN {X 0,Y 601.725,Z 315.54,A -85,B 0,C 180,E1 -774.844,E2 -774.844} C_VEL
LIN {X 0,Y 601.699,Z 330.943,A -85,B 0,C 180,E1 -777.897,E2 -777.897} C_VEL
LIN {X 0,Y 601.719,Z 340.809,A -85,B 0,C 180,E1 -779.853,E2 -779.853} C_VEL
LIN {X 0,Y 601.664,Z 354.543,A -85,B 0,C 180,E1 -782.592,E2 -782.592} C_VEL
LIN {X 0,Y 601.605,Z 367.584,A -85,B 0,C 180,E1 -785.131,E2 -785.131} C_VEL
LIN {X 0,Y 601.534,Z 381.069,A -85,B 0,C 180,E1 -787.703,E2 -787.703} C_VEL
LIN {X 0,Y 601.498,Z 394.359,A -85,B 0,C 180,E1 -790.195,E2 -790.195} C_VEL
LIN {X 0,Y 601.459,Z 407.746,A -85,B 0,C 180,E1 -792.665,E2 -792.665} C_VEL
LIN {X 0,Y 601.456,Z 423.532,A -85,B 0,C 180,E1 -795.524,E2 -795.524} C_VEL
LIN {X 0,Y 601.634,Z 425.084,A -85,B 0,C 180,E1 -795.606,E2 -795.606} C_VEL
LIN {X 0,Y 601.733,Z 440.542,A -85,B 0,C 180,E1 -795.867,E2 -795.867} C_VEL
LIN {X 0,Y 601.678,Z 453.85,A -85,B 0,C 180,E1 -796.218,E2 -796.218} C_VEL
LIN {X 0,Y 601.646,Z 466.189,A -85,B 0,C 180,E1 -796.662,E2 -796.662} C_VEL
LIN {X 0,Y 601.579,Z 479.083,A -85,B 0,C 180,E1 -797.262,E2 -797.262} C_VEL
LIN {X 0,Y 601.531,Z 492.159,A -85,B 0,C 180,E1 -798.032,E2 -798.032} C_VEL
LIN {X 0,Y 601.5,Z 503.221,A -85,B 0,C 180,E1 -798.831,E2 -798.831} C_VEL
LIN {X 0,Y 601.445,Z 513.622,A -85,B 0,C 180,E1 -799.736,E2 -799.736} C_VEL
LIN {X 0,Y 601.428,Z 523.344,A -85,B 0,C 180,E1 -800.755,E2 -800.755} C_VEL
LIN {X 0,Y 601.4,Z 531.411,A -85,B 0,C 180,E1 -801.77,E2 -801.77} C_VEL
LIN {X 0,Y 601.374,Z 539.14,A -85,B 0,C 180,E1 -802.952,E2 -802.952} C_VEL
LIN {X 0,Y 601.359,Z 544.53,A -85,B 0,C 180,E1 -803.963,E2 -803.963} C_VEL
LIN {X 0,Y 601.333,Z 550.201,A -85,B 0,C 180,E1 -805.308,E2 -805.308} C_VEL
LIN {X 0,Y 601.339,Z 554.317,A -85,B 0,C 180,E1 -806.651,E2 -806.651} C_VEL
LIN {X 0,Y 601.343,Z 557,A -85,B 0,C 180,E1 -807.991,E2 -807.991} C_VEL
LIN {X 0,Y 601.337,Z 558.332,A -85,B 0,C 180,E1 -809.331,E2 -809.331} C_VEL
LIN {X 0,Y 601.337,Z 558.331,A -85,B 0,C 180,E1 -810.67,E2 -810.67} C_VEL
LIN {X 0,Y 601.343,Z 556.999,A -85,B 0,C 180,E1 -812.01,E2 -812.01} C_VEL
LIN {X 0,Y 601.34,Z 554.314,A -85,B 0,C 180,E1 -813.351,E2 -813.351} C_VEL
LIN {X 0,Y 601.333,Z 550.196,A -85,B 0,C 180,E1 -814.693,E2 -814.693} C_VEL
LIN {X 0,Y 601.359,Z 544.524,A -85,B 0,C 180,E1 -816.038,E2 -816.038} C_VEL
LIN {X 0,Y 601.387,Z 538.122,A -85,B 0,C 180,E1 -817.218,E2 -817.218} C_VEL
LIN {X 0,Y 601.385,Z 530.165,A -85,B 0,C 180,E1 -818.4,E2 -818.4} C_VEL
LIN {X 0,Y 601.423,Z 521.845,A -85,B 0,C 180,E1 -819.416,E2 -819.416} C_VEL
LIN {X 0,Y 601.463,Z 511.832,A -85,B 0,C 180,E1 -820.435,E2 -820.435} C_VEL
LIN {X 0,Y 601.517,Z 501.43,A -85,B 0,C 180,E1 -821.312,E2 -821.312} C_VEL
LIN {X 0,Y 601.553,Z 489.496,A -85,B 0,C 180,E1 -822.14,E2 -822.14} C_VEL
LIN {X 0,Y 601.599,Z 477.371,A -85,B 0,C 180,E1 -822.825,E2 -822.825} C_VEL
LIN {X 0,Y 601.663,Z 463.939,A -85,B 0,C 180,E1 -823.425,E2 -823.425} C_VEL
LIN {X 0,Y 601.694,Z 449.759,A -85,B 0,C 180,E1 -823.901,E2 -823.901} C_VEL
LIN {X 0,Y 601.716,Z 435.434,A -85,B 0,C 180,E1 -824.234,E2 -824.234} C_VEL
LIN {X 0,Y 601.546,Z 424.567,A -85,B 0,C 180,E1 -824.406,E2 -824.406} C_VEL
LIN {X 0,Y 601.429,Z 423.353,A -85,B 0,C 180,E1 -824.503,E2 -824.503} C_VEL
LIN {X 0,Y 601.444,Z 409.652,A -85,B 0,C 180,E1 -826.986,E2 -826.986} C_VEL
LIN {X 0,Y 601.493,Z 396.264,A -85,B 0,C 180,E1 -829.452,E2 -829.452} C_VEL
LIN {X 0,Y 601.538,Z 381.062,A -85,B 0,C 180,E1 -832.298,E2 -832.298} C_VEL
LIN {X 0,Y 601.607,Z 367.577,A -85,B 0,C 180,E1 -834.87,E2 -834.87} C_VEL
LIN {X 0,Y 601.67,Z 353.66,A -85,B 0,C 180,E1 -837.582,E2 -837.582} C_VEL
LIN {X 0,Y 601.76,Z 338.892,A -85,B 0,C 180,E1 -840.533,E2 -840.533} C_VEL
LIN {X 0,Y 601.696,Z 331.78,A -85,B 0,C 180,E1 -841.907,E2 -841.907} C_VEL
LIN {X 0,Y 601.492,Z 311.644,A -85,B 0,C 180,E1 -845.402,E2 -845.402} C_VEL
LIN {X 0,Y 601.519,Z 298.762,A -85,B 0,C 180,E1 -847.73,E2 -847.73} C_VEL
LIN {X 0,Y 601.442,Z 298.307,A -85,B 0,C 180,E1 -847.842,E2 -847.842} C_VEL
LIN {X 0,Y 601.417,Z 298.19,A -85,B 0,C 180,E1 -850.573,E2 -850.573} C_VEL
LIN {X 0,Y 601.453,Z 298.195,A -85,B 0,C 180,E1 -853.584,E2 -853.584} C_VEL
LIN {X 0,Y 601.431,Z 298.188,A -85,B 0,C 180,E1 -856.428,E2 -856.428} C_VEL
LIN {X 0,Y 601.42,Z 298.197,A -85,B 0,C 180,E1 -859.427,E2 -859.427} C_VEL
LIN {X 0,Y 601.426,Z 298.195,A -85,B 0,C 180,E1 -861.732,E2 -861.732} C_VEL
LIN {X 0,Y 601.41,Z 298.19,A -85,B 0,C 180,E1 -864.247,E2 -864.247} C_VEL
LIN {X 0,Y 601.42,Z 298.189,A -85,B 0,C 180,E1 -866.686,E2 -866.686} C_VEL
LIN {X 0,Y 601.419,Z 298.193,A -85,B 0,C 180,E1 -869.058,E2 -869.058} C_VEL
LIN {X 0,Y 601.437,Z 298.197,A -85,B 0,C 180,E1 -871.374,E2 -871.374} C_VEL
LIN {X 0,Y 601.405,Z 298.196,A -85,B 0,C 180,E1 -873.636,E2 -873.636} C_VEL
LIN {X 0,Y 601.422,Z 298.189,A -85,B 0,C 180,E1 -876.59,E2 -876.59} C_VEL
LIN {X 0,Y 601.435,Z 298.194,A -85,B 0,C 180,E1 -879.478,E2 -879.478} C_VEL
LIN {X 0,Y 601.398,Z 298.192,A -85,B 0,C 180,E1 -882.312,E2 -882.312} C_VEL
LIN {X 0,Y 601.456,Z 298.334,A -85,B 0,C 180,E1 -884.996,E2 -884.996} C_VEL
LIN {X 0,Y 601.579,Z 299.092,A -85,B 0,C 180,E1 -885.107,E2 -885.107} C_VEL
LIN {X 0,Y 601.67,Z 315.281,A -85,B 0,C 180,E1 -885.671,E2 -885.671} C_VEL
LIN {X 0,Y 601.596,Z 328.601,A -85,B 0,C 180,E1 -886.283,E2 -886.283} C_VEL
LIN {X 0,Y 601.545,Z 341.027,A -85,B 0,C 180,E1 -887.003,E2 -887.003} C_VEL
LIN {X 0,Y 601.498,Z 353.04,A -85,B 0,C 180,E1 -887.859,E2 -887.859} C_VEL
LIN {X 0,Y 601.462,Z 364.204,A -85,B 0,C 180,E1 -888.836,E2 -888.836} C_VEL
LIN {X 0,Y 601.425,Z 374.275,A -85,B 0,C 180,E1 -889.905,E2 -889.905} C_VEL
LIN {X 0,Y 601.389,Z 383.384,A -85,B 0,C 180,E1 -891.092,E2 -891.092} C_VEL
LIN {X 0,Y 601.384,Z 390.761,A -85,B 0,C 180,E1 -892.277,E2 -892.277} C_VEL
LIN {X 0,Y 601.357,Z 397.254,A -85,B 0,C 180,E1 -893.604,E2 -893.604} C_VEL
LIN {X 0,Y 601.337,Z 402.303,A -85,B 0,C 180,E1 -894.971,E2 -894.971} C_VEL
LIN {X 0,Y 601.34,Z 405,A -85,B 0,C 180,E1 -895.979,E2 -895.979} C_VEL
LIN {X 0,Y 601.322,Z 407.405,A -85,B 0,C 180,E1 -897.321,E2 -897.321} C_VEL
LIN {X 0,Y 601.348,Z 408.425,A -85,B 0,C 180,E1 -898.661,E2 -898.661} C_VEL
LIN {X 0,Y 601.334,Z 408.144,A -85,B 0,C 180,E1 -900,E2 -900} C_VEL
LIN {X 0,Y 601.349,Z 406.56,A -85,B 0,C 180,E1 -901.34,E2 -901.34} C_VEL
LIN {X 0,Y 601.327,Z 403.569,A -85,B 0,C 180,E1 -902.68,E2 -902.68} C_VEL
LIN {X 0,Y 601.345,Z 399.151,A -85,B 0,C 180,E1 -904.021,E2 -904.021} C_VEL
LIN {X 0,Y 601.346,Z 394.796,A -85,B 0,C 180,E1 -905.029,E2 -905.029} C_VEL
LIN {X 0,Y 601.375,Z 388.431,A -85,B 0,C 180,E1 -906.215,E2 -906.215} C_VEL
LIN {X 0,Y 601.411,Z 380.627,A -85,B 0,C 180,E1 -907.386,E2 -907.386} C_VEL
LIN {X 0,Y 601.425,Z 370.883,A -85,B 0,C 180,E1 -908.569,E2 -908.569} C_VEL
LIN {X 0,Y 601.45,Z 360.671,A -85,B 0,C 180,E1 -909.585,E2 -909.585} C_VEL
LIN {X 0,Y 601.513,Z 349.247,A -85,B 0,C 180,E1 -910.519,E2 -910.519} C_VEL
LIN {X 0,Y 601.543,Z 344.042,A -85,B 0,C 180,E1 -910.888,E2 -910.888} C_VEL
LIN {X 0,Y 600.939,Z 339.279,A -85,B 0,C 180,E1 -911.217,E2 -911.217} C_VEL
LIN {X 0,Y 598.154,Z 331.457,A -85,B 0,C 180,E1 -911.736,E2 -911.736} C_VEL
LIN {X 0,Y 595.367,Z 323.32,A -85,B 0,C 180,E1 -912.209,E2 -912.209} C_VEL
LIN {X 0,Y 594.712,Z 318.065,A -85,B 0,C 180,E1 -912.46,E2 -912.46} C_VEL
LIN {X 0,Y 594.791,Z 304.358,A -85,B 0,C 180,E1 -912.974,E2 -912.974} C_VEL
LIN {X 0,Y 594.597,Z 300.017,A -85,B 0,C 180,E1 -913.119,E2 -913.119} C_VEL
LIN {X 0,Y 594.427,Z 299.186,A -85,B 0,C 180,E1 -913.243,E2 -913.243} C_VEL
LIN {X 0,Y 594.369,Z 299.068,A -85,B 0,C 180,E1 -915.781,E2 -915.781} C_VEL
LIN {X 0,Y 594.388,Z 299.072,A -85,B 0,C 180,E1 -918.618,E2 -918.618} C_VEL
LIN {X 0,Y 594.37,Z 299.068,A -85,B 0,C 180,E1 -921.503,E2 -921.503} C_VEL
LIN {X 0,Y 594.394,Z 299.069,A -85,B 0,C 180,E1 -924.446,E2 -924.446} C_VEL
LIN {X 0,Y 594.39,Z 299.075,A -85,B 0,C 180,E1 -926.7,E2 -926.7} C_VEL
LIN {X 0,Y 594.386,Z 299.07,A -85,B 0,C 180,E1 -928.999,E2 -928.999} C_VEL
LIN {X 0,Y 594.381,Z 299.065,A -85,B 0,C 180,E1 -931.643,E2 -931.643} C_VEL
LIN {X 0,Y 594.389,Z 299.075,A -85,B 0,C 180,E1 -934.58,E2 -934.58} C_VEL
LIN {X 0,Y 594.39,Z 299.066,A -85,B 0,C 180,E1 -937.087,E2 -937.087} C_VEL
LIN {X 0,Y 594.364,Z 299.068,A -85,B 0,C 180,E1 -939.773,E2 -939.773} C_VEL
LIN {X 0,Y 594.372,Z 299.075,A -85,B 0,C 180,E1 -942.376,E2 -942.376} C_VEL
LIN {X 0,Y 594.369,Z 299.067,A -85,B 0,C 180,E1 -945.191,E2 -945.191} C_VEL
LIN {X 0,Y 594.375,Z 299.067,A -85,B 0,C 180,E1 -947.625,E2 -947.625} C_VEL
LIN {X 0,Y 594.379,Z 299.076,A -85,B 0,C 180,E1 -950.319,E2 -950.319} C_VEL
LIN {X 0,Y 594.385,Z 299.066,A -85,B 0,C 180,E1 -952.913,E2 -952.913} C_VEL
LIN {X 0,Y 594.386,Z 299.069,A -85,B 0,C 180,E1 -955.862,E2 -955.862} C_VEL
LIN {X 0,Y 594.375,Z 299.07,A -85,B 0,C 180,E1 -958.65,E2 -958.65} C_VEL
LIN {X 0,Y 594.39,Z 299.064,A -85,B 0,C 180,E1 -961.042,E2 -961.042} C_VEL
LIN {X 0,Y 594.395,Z 299.071,A -85,B 0,C 180,E1 -963.976,E2 -963.976} C_VEL
LIN {X 0,Y 594.382,Z 299.072,A -85,B 0,C 180,E1 -966.295,E2 -966.295} C_VEL
LIN {X 0,Y 594.409,Z 299.062,A -85,B 0,C 180,E1 -969.224,E2 -969.224} C_VEL
LIN {X 0,Y 594.382,Z 299.074,A -85,B 0,C 180,E1 -972.095,E2 -972.095} C_VEL
LIN {X 0,Y 594.371,Z 299.073,A -85,B 0,C 180,E1 -974.219,E2 -974.219} C_VEL
LIN {X 0,Y 594.385,Z 299.069,A -85,B 0,C 180,E1 -976.321,E2 -976.321} C_VEL
LIN {X 0,Y 594.381,Z 299.066,A -85,B 0,C 180,E1 -979.094,E2 -979.094} C_VEL
LIN {X 0,Y 594.419,Z 299.071,A -85,B 0,C 180,E1 -981.843,E2 -981.843} C_VEL
LIN {X 0,Y 594.397,Z 299.064,A -85,B 0,C 180,E1 -984.572,E2 -984.572} C_VEL
LIN {X 0,Y 594.411,Z 299.064,A -85,B 0,C 180,E1 -987.289,E2 -987.289} C_VEL
LIN {X 0,Y 594.42,Z 299.066,A -85,B 0,C 180,E1 -989.999,E2 -989.999} C_VEL
LIN {X 0,Y 594.406,Z 299.062,A -85,B 0,C 180,E1 -992.71,E2 -992.71} C_VEL
LIN {X 0,Y 594.397,Z 299.07,A -85,B 0,C 180,E1 -995.427,E2 -995.427} C_VEL
LIN {X 0,Y 594.417,Z 299.063,A -85,B 0,C 180,E1 -998.156,E2 -998.156} C_VEL
LIN {X 0,Y 594.393,Z 299.066,A -85,B 0,C 180,E1 -1001.073,E2 -1001.073} C_VEL
LIN {X 0,Y 594.386,Z 299.073,A -85,B 0,C 180,E1 -1003.678,E2 -1003.678} C_VEL
LIN {X 0,Y 594.395,Z 299.064,A -85,B 0,C 180,E1 -1006.718,E2 -1006.718} C_VEL
LIN {X 0,Y 594.37,Z 299.075,A -85,B 0,C 180,E1 -1009.334,E2 -1009.334} C_VEL
LIN {X 0,Y 594.372,Z 299.076,A -85,B 0,C 180,E1 -1011.502,E2 -1011.502} C_VEL
LIN {X 0,Y 594.39,Z 299.064,A -85,B 0,C 180,E1 -1014.445,E2 -1014.445} C_VEL
LIN {X 0,Y 594.386,Z 299.066,A -85,B 0,C 180,E1 -1016.699,E2 -1016.699} C_VEL
LIN {X 0,Y 594.383,Z 299.07,A -85,B 0,C 180,E1 -1018.997,E2 -1018.997} C_VEL
LIN {X 0,Y 594.393,Z 299.068,A -85,B 0,C 180,E1 -1021.644,E2 -1021.644} C_VEL
LIN {X 0,Y 594.393,Z 299.065,A -85,B 0,C 180,E1 -1024.578,E2 -1024.578} C_VEL
LIN {X 0,Y 594.39,Z 299.068,A -85,B 0,C 180,E1 -1027.608,E2 -1027.608} C_VEL
LIN {X 0,Y 594.37,Z 299.069,A -85,B 0,C 180,E1 -1030.566,E2 -1030.566} C_VEL
LIN {X 0,Y 594.379,Z 299.072,A -85,B 0,C 180,E1 -1033.297,E2 -1033.297} C_VEL
LIN {X 0,Y 594.379,Z 299.066,A -85,B 0,C 180,E1 -1036.158,E2 -1036.158} C_VEL
LIN {X 0,Y 594.379,Z 299.073,A -85,B 0,C 180,E1 -1039.176,E2 -1039.176} C_VEL
LIN {X 0,Y 594.385,Z 299.065,A -85,B 0,C 180,E1 -1042.059,E2 -1042.059} C_VEL
LIN {X 0,Y 594.382,Z 299.071,A -85,B 0,C 180,E1 -1044.671,E2 -1044.671} C_VEL
LIN {X 0,Y 594.373,Z 299.073,A -85,B 0,C 180,E1 -1047.088,E2 -1047.088} C_VEL
LIN {X 0,Y 594.396,Z 299.064,A -85,B 0,C 180,E1 -1049.668,E2 -1049.668} C_VEL
LIN {X 0,Y 594.386,Z 299.071,A -85,B 0,C 180,E1 -1052.539,E2 -1052.539} C_VEL
LIN {X 0,Y 594.375,Z 299.076,A -85,B 0,C 180,E1 -1054.807,E2 -1054.807} C_VEL
LIN {X 0,Y 594.359,Z 299.07,A -85,B 0,C 180,E1 -1057.264,E2 -1057.264} C_VEL
LIN {X 0,Y 594.374,Z 299.067,A -85,B 0,C 180,E1 -1059.946,E2 -1059.946} C_VEL
LIN {X 0,Y 594.388,Z 299.072,A -85,B 0,C 180,E1 -1062.806,E2 -1062.806} C_VEL
LIN {X 0,Y 594.382,Z 299.066,A -85,B 0,C 180,E1 -1065.825,E2 -1065.825} C_VEL
LIN {X 0,Y 594.389,Z 299.072,A -85,B 0,C 180,E1 -1068.404,E2 -1068.404} C_VEL
LIN {X 0,Y 594.394,Z 299.065,A -85,B 0,C 180,E1 -1071.158,E2 -1071.158} C_VEL
LIN {X 0,Y 594.366,Z 299.069,A -85,B 0,C 180,E1 -1073.891,E2 -1073.891} C_VEL
LIN {X 0,Y 594.38,Z 299.073,A -85,B 0,C 180,E1 -1076.61,E2 -1076.61} C_VEL
LIN {X 0,Y 594.418,Z 299.061,A -85,B 0,C 180,E1 -1079.322,E2 -1079.322} C_VEL
LIN {X 0,Y 594.392,Z 299.069,A -85,B 0,C 180,E1 -1082.033,E2 -1082.033} C_VEL
LIN {X 0,Y 594.39,Z 299.068,A -85,B 0,C 180,E1 -1084.747,E2 -1084.747} C_VEL
LIN {X 0,Y 594.396,Z 299.064,A -85,B 0,C 180,E1 -1087.473,E2 -1087.473} C_VEL
LIN {X 0,Y 594.387,Z 299.075,A -85,B 0,C 180,E1 -1090.216,E2 -1090.216} C_VEL
LIN {X 0,Y 594.368,Z 299.067,A -85,B 0,C 180,E1 -1092.983,E2 -1092.983} C_VEL
LIN {X 0,Y 594.364,Z 299.072,A -85,B 0,C 180,E1 -1095.781,E2 -1095.781} C_VEL
LIN {X 0,Y 594.378,Z 299.068,A -85,B 0,C 180,E1 -1098.618,E2 -1098.618} C_VEL
LIN {X 0,Y 594.362,Z 299.07,A -85,B 0,C 180,E1 -1101.503,E2 -1101.503} C_VEL
LIN {X 0,Y 594.382,Z 299.069,A -85,B 0,C 180,E1 -1104.446,E2 -1104.446} C_VEL
LIN {X 0,Y 594.384,Z 299.066,A -85,B 0,C 180,E1 -1106.7,E2 -1106.7} C_VEL
LIN {X 0,Y 594.375,Z 299.066,A -85,B 0,C 180,E1 -1108.999,E2 -1108.999} C_VEL
LIN {X 0,Y 594.385,Z 299.071,A -85,B 0,C 180,E1 -1111.646,E2 -1111.646} C_VEL
LIN {X 0,Y 594.392,Z 299.065,A -85,B 0,C 180,E1 -1114.579,E2 -1114.579} C_VEL
LIN {X 0,Y 594.381,Z 299.066,A -85,B 0,C 180,E1 -1117.087,E2 -1117.087} C_VEL
LIN {X 0,Y 594.373,Z 299.077,A -85,B 0,C 180,E1 -1119.775,E2 -1119.775} C_VEL
LIN {X 0,Y 594.363,Z 299.07,A -85,B 0,C 180,E1 -1122.376,E2 -1122.376} C_VEL
LIN {X 0,Y 594.358,Z 299.072,A -85,B 0,C 180,E1 -1125.192,E2 -1125.192} C_VEL
LIN {X 0,Y 594.384,Z 299.075,A -85,B 0,C 180,E1 -1127.627,E2 -1127.627} C_VEL
LIN {X 0,Y 594.386,Z 299.067,A -85,B 0,C 180,E1 -1130.322,E2 -1130.322} C_VEL
LIN {X 0,Y 594.434,Z 299.243,A -85,B 0,C 180,E1 -1130.982,E2 -1130.982} C_VEL
LIN {X 0,Y 594.942,Z 302.372,A -85,B 0,C 180,E1 -1131.695,E2 -1131.695} C_VEL
LIN {X 0,Y 594.854,Z 314.313,A -85,B 0,C 180,E1 -1134.211,E2 -1134.211} C_VEL
LIN {X 0,Y 594.768,Z 329.427,A -85,B 0,C 180,E1 -1137.277,E2 -1137.277} C_VEL
LIN {X 0,Y 594.832,Z 343.037,A -85,B 0,C 180,E1 -1139.924,E2 -1139.924} C_VEL
LIN {X 0,Y 594.735,Z 356.109,A -85,B 0,C 180,E1 -1142.558,E2 -1142.558} C_VEL
LIN {X 0,Y 594.657,Z 369.498,A -85,B 0,C 180,E1 -1145.194,E2 -1145.194} C_VEL
LIN {X 0,Y 594.569,Z 382.884,A -85,B 0,C 180,E1 -1147.775,E2 -1147.775} C_VEL
LIN {X 0,Y 594.5,Z 398.184,A -85,B 0,C 180,E1 -1150.671,E2 -1150.671} C_VEL
LIN {X 0,Y 594.43,Z 413.484,A -85,B 0,C 180,E1 -1153.516,E2 -1153.516} C_VEL
LIN {X 0,Y 594.41,Z 423.872,A -85,B 0,C 180,E1 -1155.383,E2 -1155.383} C_VEL
LIN {X 0,Y 594.884,Z 427.658,A -85,B 0,C 180,E1 -1155.476,E2 -1155.476} C_VEL
LIN {X 0,Y 594.804,Z 441.984,A -85,B 0,C 180,E1 -1155.733,E2 -1155.733} C_VEL
LIN {X 0,Y 594.775,Z 456.201,A -85,B 0,C 180,E1 -1156.134,E2 -1156.134} C_VEL
LIN {X 0,Y 594.691,Z 470.146,A -85,B 0,C 180,E1 -1156.677,E2 -1156.677} C_VEL
LIN {X 0,Y 594.62,Z 483.79,A -85,B 0,C 180,E1 -1157.371,E2 -1157.371} C_VEL
LIN {X 0,Y 594.548,Z 495.98,A -85,B 0,C 180,E1 -1158.149,E2 -1158.149} C_VEL
LIN {X 0,Y 594.461,Z 506.808,A -85,B 0,C 180,E1 -1158.991,E2 -1158.991} C_VEL
LIN {X 0,Y 594.4,Z 517.088,A -85,B 0,C 180,E1 -1159.957,E2 -1159.957} C_VEL
LIN {X 0,Y 594.369,Z 526.204,A -85,B 0,C 180,E1 -1160.987,E2 -1160.987} C_VEL
LIN {X 0,Y 594.315,Z 534.923,A -85,B 0,C 180,E1 -1162.185,E2 -1162.185} C_VEL
LIN {X 0,Y 594.276,Z 542.138,A -85,B 0,C 180,E1 -1163.412,E2 -1163.412} C_VEL
LIN {X 0,Y 594.275,Z 547.571,A -85,B 0,C 180,E1 -1164.572,E2 -1164.572} C_VEL
LIN {X 0,Y 594.259,Z 552.444,A -85,B 0,C 180,E1 -1165.932,E2 -1165.932} C_VEL
LIN {X 0,Y 594.224,Z 555.833,A -85,B 0,C 180,E1 -1167.289,E2 -1167.289} C_VEL
LIN {X 0,Y 594.242,Z 557.832,A -85,B 0,C 180,E1 -1168.645,E2 -1168.645} C_VEL
LIN {X 0,Y 594.234,Z 558.5,A -85,B 0,C 180,E1 -1170.001,E2 -1170.001} C_VEL
LIN {X 0,Y 594.242,Z 557.831,A -85,B 0,C 180,E1 -1171.356,E2 -1171.356} C_VEL
LIN {X 0,Y 594.224,Z 555.831,A -85,B 0,C 180,E1 -1172.712,E2 -1172.712} C_VEL
LIN {X 0,Y 594.259,Z 552.44,A -85,B 0,C 180,E1 -1174.07,E2 -1174.07} C_VEL
LIN {X 0,Y 594.275,Z 547.565,A -85,B 0,C 180,E1 -1175.429,E2 -1175.429} C_VEL
LIN {X 0,Y 594.3,Z 542.031,A -85,B 0,C 180,E1 -1176.607,E2 -1176.607} C_VEL
LIN {X 0,Y 594.316,Z 534.916,A -85,B 0,C 180,E1 -1177.817,E2 -1177.817} C_VEL
LIN {X 0,Y 594.369,Z 526.194,A -85,B 0,C 180,E1 -1179.014,E2 -1179.014} C_VEL
LIN {X 0,Y 594.4,Z 517.076,A -85,B 0,C 180,E1 -1180.044,E2 -1180.044} C_VEL
LIN {X 0,Y 594.479,Z 506.696,A -85,B 0,C 180,E1 -1181.018,E2 -1181.018} C_VEL
LIN {X 0,Y 594.573,Z 494.697,A -85,B 0,C 180,E1 -1181.939,E2 -1181.939} C_VEL
LIN {X 0,Y 594.62,Z 482.202,A -85,B 0,C 180,E1 -1182.717,E2 -1182.717} C_VEL
LIN {X 0,Y 594.691,Z 470.116,A -85,B 0,C 180,E1 -1183.324,E2 -1183.324} C_VEL
LIN {X 0,Y 594.776,Z 456.184,A -85,B 0,C 180,E1 -1183.866,E2 -1183.866} C_VEL
LIN {X 0,Y 594.818,Z 442.265,A -85,B 0,C 180,E1 -1184.26,E2 -1184.26} C_VEL
LIN {X 0,Y 594.863,Z 428.53,A -85,B 0,C 180,E1 -1184.512,E2 -1184.512} C_VEL
LIN {X 0,Y 594.563,Z 424.995,A -85,B 0,C 180,E1 -1184.57,E2 -1184.57} C_VEL
LIN {X 0,Y 594.424,Z 423.589,A -85,B 0,C 180,E1 -1184.643,E2 -1184.643} C_VEL
LIN {X 0,Y 594.425,Z 407.739,A -85,B 0,C 180,E1 -1187.548,E2 -1187.548} C_VEL
LIN {X 0,Y 594.504,Z 396.264,A -85,B 0,C 180,E1 -1189.69,E2 -1189.69} C_VEL
LIN {X 0,Y 594.592,Z 381.413,A -85,B 0,C 180,E1 -1192.505,E2 -1192.505} C_VEL
LIN {X 0,Y 594.682,Z 365.665,A -85,B 0,C 180,E1 -1195.554,E2 -1195.554} C_VEL
LIN {X 0,Y 594.789,Z 350.365,A -85,B 0,C 180,E1 -1198.591,E2 -1198.591} C_VEL
LIN {X 0,Y 594.847,Z 340.636,A -85,B 0,C 180,E1 -1200.534,E2 -1200.534} C_VEL
LIN {X 0,Y 594.434,Z 324.462,A -85,B 0,C 180,E1 -1203.352,E2 -1203.352} C_VEL
LIN {X 0,Y 594.498,Z 309.42,A -85,B 0,C 180,E1 -1206.025,E2 -1206.025} C_VEL
LIN {X 0,Y 594.589,Z 300.724,A -85,B 0,C 180,E1 -1207.633,E2 -1207.633} C_VEL
LIN {X 0,Y 594.414,Z 299.154,A -85,B 0,C 180,E1 -1207.993,E2 -1207.993} C_VEL
LIN {X 0,Y 594.38,Z 299.067,A -85,B 0,C 180,E1 -1210.822,E2 -1210.822} C_VEL
LIN {X 0,Y 594.386,Z 299.072,A -85,B 0,C 180,E1 -1213.841,E2 -1213.841} C_VEL
LIN {X 0,Y 594.369,Z 299.068,A -85,B 0,C 180,E1 -1216.701,E2 -1216.701} C_VEL
LIN {X 0,Y 594.375,Z 299.075,A -85,B 0,C 180,E1 -1219.434,E2 -1219.434} C_VEL
LIN {X 0,Y 594.392,Z 299.064,A -85,B 0,C 180,E1 -1222.392,E2 -1222.392} C_VEL
LIN {X 0,Y 594.387,Z 299.065,A -85,B 0,C 180,E1 -1224.672,E2 -1224.672} C_VEL
LIN {X 0,Y 594.382,Z 299.07,A -85,B 0,C 180,E1 -1227.089,E2 -1227.089} C_VEL
LIN {X 0,Y 594.389,Z 299.07,A -85,B 0,C 180,E1 -1229.672,E2 -1229.672} C_VEL
LIN {X 0,Y 594.378,Z 299.067,A -85,B 0,C 180,E1 -1232.539,E2 -1232.539} C_VEL
LIN {X 0,Y 594.376,Z 299.069,A -85,B 0,C 180,E1 -1234.807,E2 -1234.807} C_VEL
LIN {X 0,Y 594.368,Z 299.078,A -85,B 0,C 180,E1 -1237.265,E2 -1237.265} C_VEL
LIN {X 0,Y 594.379,Z 299.067,A -85,B 0,C 180,E1 -1239.947,E2 -1239.947} C_VEL
LIN {X 0,Y 594.393,Z 299.069,A -85,B 0,C 180,E1 -1242.807,E2 -1242.807} C_VEL
LIN {X 0,Y 594.456,Z 299.302,A -85,B 0,C 180,E1 -1244.88,E2 -1244.88} C_VEL
LIN {X 0,Y 594.578,Z 300.04,A -85,B 0,C 180,E1 -1244.971,E2 -1244.971} C_VEL
LIN {X 0,Y 594.787,Z 304.098,A -85,B 0,C 180,E1 -1245.108,E2 -1245.108} C_VEL
LIN {X 0,Y 594.721,Z 318.084,A -85,B 0,C 180,E1 -1245.631,E2 -1245.631} C_VEL
LIN {X 0,Y 594.643,Z 331.077,A -85,B 0,C 180,E1 -1246.264,E2 -1246.264} C_VEL
LIN {X 0,Y 594.56,Z 343.482,A -85,B 0,C 180,E1 -1247.021,E2 -1247.021} C_VEL
LIN {X 0,Y 594.5,Z 354.997,A -85,B 0,C 180,E1 -1247.887,E2 -1247.887} C_VEL
LIN {X 0,Y 594.435,Z 364.784,A -85,B 0,C 180,E1 -1248.77,E2 -1248.77} C_VEL
LIN {X 0,Y 594.383,Z 374.178,A -85,B 0,C 180,E1 -1249.784,E2 -1249.784} C_VEL
LIN {X 0,Y 594.34,Z 383.306,A -85,B 0,C 180,E1 -1250.986,E2 -1250.986} C_VEL
LIN {X 0,Y 594.305,Z 390.696,A -85,B 0,C 180,E1 -1252.184,E2 -1252.184} C_VEL
LIN {X 0,Y 594.273,Z 396.741,A -85,B 0,C 180,E1 -1253.416,E2 -1253.416} C_VEL
LIN {X 0,Y 594.27,Z 401.166,A -85,B 0,C 180,E1 -1254.571,E2 -1254.571} C_VEL
LIN {X 0,Y 594.253,Z 404.975,A -85,B 0,C 180,E1 -1255.931,E2 -1255.931} C_VEL
LIN {X 0,Y 594.223,Z 407.388,A -85,B 0,C 180,E1 -1257.289,E2 -1257.289} C_VEL
LIN {X 0,Y 594.247,Z 408.423,A -85,B 0,C 180,E1 -1258.645,E2 -1258.645} C_VEL
LIN {X 0,Y 594.235,Z 408.151,A -85,B 0,C 180,E1 -1260,E2 -1260} C_VEL
LIN {X 0,Y 594.249,Z 406.58,A -85,B 0,C 180,E1 -1261.356,E2 -1261.356} C_VEL
LIN {X 0,Y 594.23,Z 403.602,A -85,B 0,C 180,E1 -1262.712,E2 -1262.712} C_VEL
LIN {X 0,Y 594.261,Z 399.196,A -85,B 0,C 180,E1 -1264.069,E2 -1264.069} C_VEL
LIN {X 0,Y 594.256,Z 394.852,A -85,B 0,C 180,E1 -1265.089,E2 -1265.089} C_VEL
LIN {X 0,Y 594.317,Z 387.86,A -85,B 0,C 180,E1 -1266.398,E2 -1266.398} C_VEL
LIN {X 0,Y 594.34,Z 380.716,A -85,B 0,C 180,E1 -1267.474,E2 -1267.474} C_VEL
LIN {X 0,Y 594.377,Z 370.988,A -85,B 0,C 180,E1 -1268.671,E2 -1268.671} C_VEL
LIN {X 0,Y 594.425,Z 360.803,A -85,B 0,C 180,E1 -1269.7,E2 -1269.7} C_VEL
LIN {X 0,Y 594.524,Z 349.401,A -85,B 0,C 180,E1 -1270.644,E2 -1270.644} C_VEL
LIN {X 0,Y 594.597,Z 337.766,A -85,B 0,C 180,E1 -1271.439,E2 -1271.439} C_VEL
LIN {X 0,Y 594.679,Z 325.65,A -85,B 0,C 180,E1 -1272.109,E2 -1272.109} C_VEL
LIN {X 0,Y 594.712,Z 318.065,A -85,B 0,C 180,E1 -1272.46,E2 -1272.46} C_VEL
LIN {X 0,Y 594.205,Z 311.626,A -85,B 0,C 180,E1 -1272.753,E2 -1272.753} C_VEL
LIN {X 0,Y 592.554,Z 307.341,A -85,B 0,C 180,E1 -1272.927,E2 -1272.927} C_VEL
LIN {X 0,Y 590.17,Z 303.571,A -85,B 0,C 180,E1 -1273.108,E2 -1273.108} C_VEL
LIN {X 0,Y 587.48,Z 300.473,A -85,B 0,C 180,E1 -1273.305,E2 -1273.305} C_VEL
LIN {X 0,Y 587.393,Z 300.245,A -85,B 0,C 180,E1 -1273.34,E2 -1273.34} C_VEL
LIN {X 0,Y 587.363,Z 299.942,A -85,B 0,C 180,E1 -1273.846,E2 -1273.846} C_VEL
LIN {X 0,Y 587.366,Z 299.949,A -85,B 0,C 180,E1 -1276.818,E2 -1276.818} C_VEL
LIN {X 0,Y 587.347,Z 299.943,A -85,B 0,C 180,E1 -1279.575,E2 -1279.575} C_VEL
LIN {X 0,Y 587.344,Z 299.948,A -85,B 0,C 180,E1 -1282.514,E2 -1282.514} C_VEL
LIN {X 0,Y 587.355,Z 299.951,A -85,B 0,C 180,E1 -1284.759,E2 -1284.759} C_VEL
LIN {X 0,Y 587.356,Z 299.94,A -85,B 0,C 180,E1 -1287.693,E2 -1287.693} C_VEL
LIN {X 0,Y 587.341,Z 299.95,A -85,B 0,C 180,E1 -1290.51,E2 -1290.51} C_VEL
LIN {X 0,Y 587.338,Z 299.943,A -85,B 0,C 180,E1 -1293.397,E2 -1293.397} C_VEL
LIN {X 0,Y 587.324,Z 299.946,A -85,B 0,C 180,E1 -1295.898,E2 -1295.898} C_VEL
LIN {X 0,Y 587.335,Z 299.953,A -85,B 0,C 180,E1 -1298.479,E2 -1298.479} C_VEL
LIN {X 0,Y 587.34,Z 299.944,A -85,B 0,C 180,E1 -1301.157,E2 -1301.157} C_VEL
LIN {X 0,Y 587.332,Z 299.948,A -85,B 0,C 180,E1 -1304.113,E2 -1304.113} C_VEL
LIN {X 0,Y 587.327,Z 299.946,A -85,B 0,C 180,E1 -1306.994,E2 -1306.994} C_VEL
LIN {X 0,Y 587.318,Z 299.947,A -85,B 0,C 180,E1 -1309.746,E2 -1309.746} C_VEL
LIN {X 0,Y 587.349,Z 299.95,A -85,B 0,C 180,E1 -1312.392,E2 -1312.392} C_VEL
LIN {X 0,Y 587.366,Z 299.942,A -85,B 0,C 180,E1 -1315.78,E2 -1315.78} C_VEL
LIN {X 0,Y 587.348,Z 299.952,A -85,B 0,C 180,E1 -1318.231,E2 -1318.231} C_VEL
LIN {X 0,Y 587.357,Z 299.941,A -85,B 0,C 180,E1 -1320.866,E2 -1320.866} C_VEL
LIN {X 0,Y 587.367,Z 299.944,A -85,B 0,C 180,E1 -1323.819,E2 -1323.819} C_VEL
LIN {X 0,Y 587.336,Z 299.951,A -85,B 0,C 180,E1 -1325.993,E2 -1325.993} C_VEL
LIN {X 0,Y 587.328,Z 299.952,A -85,B 0,C 180,E1 -1328.225,E2 -1328.225} C_VEL
LIN {X 0,Y 587.355,Z 299.941,A -85,B 0,C 180,E1 -1331.151,E2 -1331.151} C_VEL
LIN {X 0,Y 587.356,Z 299.941,A -85,B 0,C 180,E1 -1333.311,E2 -1333.311} C_VEL
LIN {X 0,Y 587.364,Z 299.946,A -85,B 0,C 180,E1 -1336.154,E2 -1336.154} C_VEL
LIN {X 0,Y 587.347,Z 299.942,A -85,B 0,C 180,E1 -1338.962,E2 -1338.962} C_VEL
LIN {X 0,Y 587.371,Z 299.947,A -85,B 0,C 180,E1 -1341.744,E2 -1341.744} C_VEL
LIN {X 0,Y 587.364,Z 299.941,A -85,B 0,C 180,E1 -1344.507,E2 -1344.507} C_VEL
LIN {X 0,Y 587.377,Z 299.94,A -85,B 0,C 180,E1 -1347.256,E2 -1347.256} C_VEL
LIN {X 0,Y 587.389,Z 299.942,A -85,B 0,C 180,E1 -1349.999,E2 -1349.999} C_VEL
LIN {X 0,Y 587.373,Z 299.938,A -85,B 0,C 180,E1 -1352.743,E2 -1352.743} C_VEL
LIN {X 0,Y 587.362,Z 299.947,A -85,B 0,C 180,E1 -1355.492,E2 -1355.492} C_VEL
LIN {X 0,Y 587.369,Z 299.94,A -85,B 0,C 180,E1 -1358.255,E2 -1358.255} C_VEL
LIN {X 0,Y 587.353,Z 299.944,A -85,B 0,C 180,E1 -1361.133,E2 -1361.133} C_VEL
LIN {X 0,Y 587.369,Z 299.94,A -85,B 0,C 180,E1 -1364.26,E2 -1364.26} C_VEL
LIN {X 0,Y 587.353,Z 299.95,A -85,B 0,C 180,E1 -1367.405,E2 -1367.405} C_VEL
LIN {X 0,Y 587.331,Z 299.944,A -85,B 0,C 180,E1 -1370.304,E2 -1370.304} C_VEL
LIN {X 0,Y 587.324,Z 299.953,A -85,B 0,C 180,E1 -1373.258,E2 -1373.258} C_VEL
LIN {X 0,Y 587.338,Z 299.95,A -85,B 0,C 180,E1 -1375.516,E2 -1375.516} C_VEL
LIN {X 0,Y 587.348,Z 299.944,A -85,B 0,C 180,E1 -1377.817,E2 -1377.817} C_VEL
LIN {X 0,Y 587.342,Z 299.943,A -85,B 0,C 180,E1 -1380.51,E2 -1380.51} C_VEL
LIN {X 0,Y 587.341,Z 299.95,A -85,B 0,C 180,E1 -1383.111,E2 -1383.111} C_VEL
LIN {X 0,Y 587.3,Z 299.952,A -85,B 0,C 180,E1 -1385.537,E2 -1385.537} C_VEL
LIN {X 0,Y 587.34,Z 299.944,A -85,B 0,C 180,E1 -1387.838,E2 -1387.838} C_VEL
LIN {X 0,Y 587.317,Z 299.945,A -85,B 0,C 180,E1 -1390.253,E2 -1390.253} C_VEL
LIN {X 0,Y 587.325,Z 299.954,A -85,B 0,C 180,E1 -1393.119,E2 -1393.119} C_VEL
LIN {X 0,Y 587.331,Z 299.943,A -85,B 0,C 180,E1 -1396.05,E2 -1396.05} C_VEL
LIN {X 0,Y 587.335,Z 299.952,A -85,B 0,C 180,E1 -1398.924,E2 -1398.924} C_VEL
LIN {X 0,Y 587.331,Z 299.946,A -85,B 0,C 180,E1 -1401.52,E2 -1401.52} C_VEL
LIN {X 0,Y 587.349,Z 299.944,A -85,B 0,C 180,E1 -1404.454,E2 -1404.454} C_VEL
LIN {X 0,Y 587.335,Z 299.954,A -85,B 0,C 180,E1 -1406.887,E2 -1406.887} C_VEL
LIN {X 0,Y 587.347,Z 299.943,A -85,B 0,C 180,E1 -1409.487,E2 -1409.487} C_VEL
LIN {X 0,Y 587.346,Z 299.944,A -85,B 0,C 180,E1 -1412.306,E2 -1412.306} C_VEL
LIN {X 0,Y 587.333,Z 299.949,A -85,B 0,C 180,E1 -1414.483,E2 -1414.483} C_VEL
LIN {X 0,Y 587.313,Z 299.95,A -85,B 0,C 180,E1 -1417.13,E2 -1417.13} C_VEL
LIN {X 0,Y 587.327,Z 299.944,A -85,B 0,C 180,E1 -1419.695,E2 -1419.695} C_VEL
LIN {X 0,Y 587.355,Z 299.95,A -85,B 0,C 180,E1 -1422.594,E2 -1422.594} C_VEL
LIN {X 0,Y 587.358,Z 299.94,A -85,B 0,C 180,E1 -1425.739,E2 -1425.739} C_VEL
LIN {X 0,Y 587.337,Z 299.948,A -85,B 0,C 180,E1 -1428.263,E2 -1428.263} C_VEL
LIN {X 0,Y 587.34,Z 299.945,A -85,B 0,C 180,E1 -1431.051,E2 -1431.051} C_VEL
LIN {X 0,Y 587.368,Z 299.939,A -85,B 0,C 180,E1 -1433.263,E2 -1433.263} C_VEL
LIN {X 0,Y 587.312,Z 299.948,A -85,B 0,C 180,E1 -1435.883,E2 -1435.883} C_VEL
LIN {X 0,Y 587.363,Z 299.943,A -85,B 0,C 180,E1 -1437.943,E2 -1437.943} C_VEL
LIN {X 0,Y 587.389,Z 299.941,A -85,B 0,C 180,E1 -1440.685,E2 -1440.685} C_VEL
LIN {X 0,Y 587.33,Z 299.944,A -85,B 0,C 180,E1 -1443.43,E2 -1443.43} C_VEL
LIN {X 0,Y 587.355,Z 299.941,A -85,B 0,C 180,E1 -1445.493,E2 -1445.493} C_VEL
LIN {X 0,Y 587.364,Z 299.95,A -85,B 0,C 180,E1 -1448.255,E2 -1448.255} C_VEL
LIN {X 0,Y 587.339,Z 299.943,A -85,B 0,C 180,E1 -1451.134,E2 -1451.134} C_VEL
LIN {X 0,Y 587.355,Z 299.945,A -85,B 0,C 180,E1 -1453.846,E2 -1453.846} C_VEL
LIN {X 0,Y 587.355,Z 299.941,A -85,B 0,C 180,E1 -1456.819,E2 -1456.819} C_VEL
LIN {X 0,Y 587.339,Z 299.945,A -85,B 0,C 180,E1 -1459.575,E2 -1459.575} C_VEL
LIN {X 0,Y 587.334,Z 299.946,A -85,B 0,C 180,E1 -1462.514,E2 -1462.514} C_VEL
LIN {X 0,Y 587.345,Z 299.942,A -85,B 0,C 180,E1 -1464.759,E2 -1464.759} C_VEL
LIN {X 0,Y 587.333,Z 299.943,A -85,B 0,C 180,E1 -1467.046,E2 -1467.046} C_VEL
LIN {X 0,Y 587.344,Z 299.944,A -85,B 0,C 180,E1 -1469.38,E2 -1469.38} C_VEL
LIN {X 0,Y 587.348,Z 299.951,A -85,B 0,C 180,E1 -1471.838,E2 -1471.838} C_VEL
LIN {X 0,Y 587.351,Z 299.944,A -85,B 0,C 180,E1 -1474.35,E2 -1474.35} C_VEL
LIN {X 0,Y 587.347,Z 299.942,A -85,B 0,C 180,E1 -1476.747,E2 -1476.747} C_VEL
LIN {X 0,Y 587.342,Z 299.946,A -85,B 0,C 180,E1 -1479.36,E2 -1479.36} C_VEL
LIN {X 0,Y 587.329,Z 299.949,A -85,B 0,C 180,E1 -1482.108,E2 -1482.108} C_VEL
LIN {X 0,Y 587.31,Z 299.949,A -85,B 0,C 180,E1 -1485.089,E2 -1485.089} C_VEL
LIN {X 0,Y 587.348,Z 299.95,A -85,B 0,C 180,E1 -1487.928,E2 -1487.928} C_VEL
LIN {X 0,Y 587.371,Z 300.105,A -85,B 0,C 180,E1 -1490.706,E2 -1490.706} C_VEL
LIN {X 0,Y 588.113,Z 305.195,A -85,B 0,C 180,E1 -1491.873,E2 -1491.873} C_VEL
LIN {X 0,Y 587.931,Z 318.445,A -85,B 0,C 180,E1 -1494.68,E2 -1494.68} C_VEL
LIN {X 0,Y 587.853,Z 332.003,A -85,B 0,C 180,E1 -1497.454,E2 -1497.454} C_VEL
LIN {X 0,Y 587.893,Z 346.292,A -85,B 0,C 180,E1 -1500.258,E2 -1500.258} C_VEL
LIN {X 0,Y 587.826,Z 358.038,A -85,B 0,C 180,E1 -1502.598,E2 -1502.598} C_VEL
LIN {X 0,Y 587.701,Z 371.855,A -85,B 0,C 180,E1 -1505.346,E2 -1505.346} C_VEL
LIN {X 0,Y 587.565,Z 386.709,A -85,B 0,C 180,E1 -1508.236,E2 -1508.236} C_VEL
LIN {X 0,Y 587.493,Z 402.009,A -85,B 0,C 180,E1 -1511.157,E2 -1511.157} C_VEL
LIN {X 0,Y 587.361,Z 417.309,A -85,B 0,C 180,E1 -1514.027,E2 -1514.027} C_VEL
LIN {X 0,Y 587.399,Z 423.869,A -85,B 0,C 180,E1 -1515.205,E2 -1515.205} C_VEL
LIN {X 0,Y 588.01,Z 427.418,A -85,B 0,C 180,E1 -1515.298,E2 -1515.298} C_VEL
LIN {X 0,Y 587.933,Z 441.754,A -85,B 0,C 180,E1 -1515.557,E2 -1515.557} C_VEL
LIN {X 0,Y 587.895,Z 454.633,A -85,B 0,C 180,E1 -1515.915,E2 -1515.915} C_VEL
LIN {X 0,Y 587.779,Z 468.178,A -85,B 0,C 180,E1 -1516.43,E2 -1516.43} C_VEL
LIN {X 0,Y 587.672,Z 480.659,A -85,B 0,C 180,E1 -1517.043,E2 -1517.043} C_VEL
LIN {X 0,Y 587.579,Z 493.44,A -85,B 0,C 180,E1 -1517.831,E2 -1517.831} C_VEL
LIN {X 0,Y 587.469,Z 505.09,A -85,B 0,C 180,E1 -1518.715,E2 -1518.715} C_VEL
LIN {X 0,Y 587.372,Z 515.398,A -85,B 0,C 180,E1 -1519.661,E2 -1519.661} C_VEL
LIN {X 0,Y 587.33,Z 524.829,A -85,B 0,C 180,E1 -1520.704,E2 -1520.704} C_VEL
LIN {X 0,Y 587.268,Z 533.803,A -85,B 0,C 180,E1 -1521.917,E2 -1521.917} C_VEL
LIN {X 0,Y 587.208,Z 541.056,A -85,B 0,C 180,E1 -1523.127,E2 -1523.127} C_VEL
LIN {X 0,Y 587.227,Z 546.139,A -85,B 0,C 180,E1 -1524.162,E2 -1524.162} C_VEL
LIN {X 0,Y 587.185,Z 551.385,A -85,B 0,C 180,E1 -1525.539,E2 -1525.539} C_VEL
LIN {X 0,Y 587.182,Z 554.317,A -85,B 0,C 180,E1 -1526.57,E2 -1526.57} C_VEL
LIN {X 0,Y 587.14,Z 557.001,A -85,B 0,C 180,E1 -1527.943,E2 -1527.943} C_VEL
LIN {X 0,Y 587.137,Z 558.333,A -85,B 0,C 180,E1 -1529.315,E2 -1529.315} C_VEL
LIN {X 0,Y 587.137,Z 558.332,A -85,B 0,C 180,E1 -1530.686,E2 -1530.686} C_VEL
LIN {X 0,Y 587.14,Z 557,A -85,B 0,C 180,E1 -1532.059,E2 -1532.059} C_VEL
LIN {X 0,Y 587.182,Z 554.315,A -85,B 0,C 180,E1 -1533.432,E2 -1533.432} C_VEL
LIN {X 0,Y 587.141,Z 550.197,A -85,B 0,C 180,E1 -1534.807,E2 -1534.807} C_VEL
LIN {X 0,Y 587.227,Z 546.133,A -85,B 0,C 180,E1 -1535.839,E2 -1535.839} C_VEL
LIN {X 0,Y 587.226,Z 539.134,A -85,B 0,C 180,E1 -1537.22,E2 -1537.22} C_VEL
LIN {X 0,Y 587.277,Z 531.404,A -85,B 0,C 180,E1 -1538.43,E2 -1538.43} C_VEL
LIN {X 0,Y 587.336,Z 523.334,A -85,B 0,C 180,E1 -1539.471,E2 -1539.471} C_VEL
LIN {X 0,Y 587.402,Z 513.609,A -85,B 0,C 180,E1 -1540.514,E2 -1540.514} C_VEL
LIN {X 0,Y 587.508,Z 502.821,A -85,B 0,C 180,E1 -1541.471,E2 -1541.471} C_VEL
LIN {X 0,Y 587.606,Z 490.853,A -85,B 0,C 180,E1 -1542.345,E2 -1542.345} C_VEL
LIN {X 0,Y 587.694,Z 479.058,A -85,B 0,C 180,E1 -1543.046,E2 -1543.046} C_VEL
LIN {X 0,Y 587.816,Z 466.155,A -85,B 0,C 180,E1 -1543.659,E2 -1543.659} C_VEL
LIN {X 0,Y 587.905,Z 451.784,A -85,B 0,C 180,E1 -1544.175,E2 -1544.175} C_VEL
LIN {X 0,Y 587.967,Z 438.059,A -85,B 0,C 180,E1 -1544.523,E2 -1544.523} C_VEL
LIN {X 0,Y 587.827,Z 426.562,A -85,B 0,C 180,E1 -1544.719,E2 -1544.719} C_VEL
LIN {X 0,Y 587.399,Z 423.848,A -85,B 0,C 180,E1 -1544.796,E2 -1544.796} C_VEL
LIN {X 0,Y 587.394,Z 409.652,A -85,B 0,C 180,E1 -1547.405,E2 -1547.405} C_VEL
LIN {X 0,Y 587.502,Z 396.264,A -85,B 0,C 180,E1 -1549.934,E2 -1549.934} C_VEL
LIN {X 0,Y 587.62,Z 381.757,A -85,B 0,C 180,E1 -1552.72,E2 -1552.72} C_VEL
LIN {X 0,Y 587.731,Z 367.577,A -85,B 0,C 180,E1 -1555.499,E2 -1555.499} C_VEL
LIN {X 0,Y 587.845,Z 354.19,A -85,B 0,C 180,E1 -1558.18,E2 -1558.18} C_VEL
LIN {X 0,Y 587.886,Z 347.195,A -85,B 0,C 180,E1 -1559.547,E2 -1559.547} C_VEL
LIN {X 0,Y 587.592,Z 332.064,A -85,B 0,C 180,E1 -1562.191,E2 -1562.191} C_VEL
LIN {X 0,Y 587.482,Z 313.236,A -85,B 0,C 180,E1 -1565.563,E2 -1565.563} C_VEL
LIN {X 0,Y 587.628,Z 302.436,A -85,B 0,C 180,E1 -1567.587,E2 -1567.587} C_VEL
LIN {X 0,Y 587.371,Z 300.053,A -85,B 0,C 180,E1 -1568.093,E2 -1568.093} C_VEL
LIN {X 0,Y 587.339,Z 299.946,A -85,B 0,C 180,E1 -1571.075,E2 -1571.075} C_VEL
LIN {X 0,Y 587.338,Z 299.946,A -85,B 0,C 180,E1 -1574.114,E2 -1574.114} C_VEL
LIN {X 0,Y 587.318,Z 299.948,A -85,B 0,C 180,E1 -1576.994,E2 -1576.994} C_VEL
LIN {X 0,Y 587.322,Z 299.952,A -85,B 0,C 180,E1 -1579.746,E2 -1579.746} C_VEL
LIN {X 0,Y 587.348,Z 299.942,A -85,B 0,C 180,E1 -1582.393,E2 -1582.393} C_VEL
LIN {X 0,Y 587.353,Z 299.944,A -85,B 0,C 180,E1 -1584.946,E2 -1584.946} C_VEL
LIN {X 0,Y 587.342,Z 299.953,A -85,B 0,C 180,E1 -1587.421,E2 -1587.421} C_VEL
LIN {X 0,Y 587.336,Z 299.947,A -85,B 0,C 180,E1 -1589.83,E2 -1589.83} C_VEL
LIN {X 0,Y 587.355,Z 299.941,A -85,B 0,C 180,E1 -1592.307,E2 -1592.307} C_VEL
LIN {X 0,Y 587.354,Z 299.951,A -85,B 0,C 180,E1 -1595.242,E2 -1595.242} C_VEL
LIN {X 0,Y 587.325,Z 299.945,A -85,B 0,C 180,E1 -1598.226,E2 -1598.226} C_VEL
LIN {X 0,Y 587.354,Z 299.951,A -85,B 0,C 180,E1 -1601.151,E2 -1601.151} C_VEL
LIN {X 0,Y 587.328,Z 299.947,A -85,B 0,C 180,E1 -1604.025,E2 -1604.025} C_VEL
LIN {X 0,Y 587.384,Z 300.206,A -85,B 0,C 180,E1 -1604.738,E2 -1604.738} C_VEL
LIN {X 0,Y 587.573,Z 300.987,A -85,B 0,C 180,E1 -1604.832,E2 -1604.832} C_VEL
LIN {X 0,Y 587.88,Z 303.677,A -85,B 0,C 180,E1 -1604.929,E2 -1604.929} C_VEL
LIN {X 0,Y 587.819,Z 316.813,A -85,B 0,C 180,E1 -1605.415,E2 -1605.415} C_VEL
LIN {X 0,Y 587.713,Z 329.904,A -85,B 0,C 180,E1 -1606.047,E2 -1606.047} C_VEL
LIN {X 0,Y 587.573,Z 342.01,A -85,B 0,C 180,E1 -1606.776,E2 -1606.776} C_VEL
LIN {X 0,Y 587.471,Z 353.806,A -85,B 0,C 180,E1 -1607.653,E2 -1607.653} C_VEL
LIN {X 0,Y 587.401,Z 364.472,A -85,B 0,C 180,E1 -1608.615,E2 -1608.615} C_VEL
LIN {X 0,Y 587.353,Z 374.08,A -85,B 0,C 180,E1 -1609.66,E2 -1609.66} C_VEL
LIN {X 0,Y 587.269,Z 383.228,A -85,B 0,C 180,E1 -1610.876,E2 -1610.876} C_VEL
LIN {X 0,Y 587.219,Z 390.631,A -85,B 0,C 180,E1 -1612.089,E2 -1612.089} C_VEL
LIN {X 0,Y 587.196,Z 397.032,A -85,B 0,C 180,E1 -1613.418,E2 -1613.418} C_VEL
LIN {X 0,Y 587.193,Z 401.131,A -85,B 0,C 180,E1 -1614.506,E2 -1614.506} C_VEL
LIN {X 0,Y 587.169,Z 404.95,A -85,B 0,C 180,E1 -1615.882,E2 -1615.882} C_VEL
LIN {X 0,Y 587.129,Z 407.371,A -85,B 0,C 180,E1 -1617.256,E2 -1617.256} C_VEL
LIN {X 0,Y 587.147,Z 408.42,A -85,B 0,C 180,E1 -1618.628,E2 -1618.628} C_VEL
LIN {X 0,Y 587.135,Z 408.159,A -85,B 0,C 180,E1 -1620,E2 -1620} C_VEL
LIN {X 0,Y 587.148,Z 406.599,A -85,B 0,C 180,E1 -1621.372,E2 -1621.372} C_VEL
LIN {X 0,Y 587.137,Z 403.636,A -85,B 0,C 180,E1 -1622.745,E2 -1622.745} C_VEL
LIN {X 0,Y 587.182,Z 399.241,A -85,B 0,C 180,E1 -1624.118,E2 -1624.118} C_VEL
LIN {X 0,Y 587.21,Z 393.27,A -85,B 0,C 180,E1 -1625.495,E2 -1625.495} C_VEL
LIN {X 0,Y 587.207,Z 387.236,A -85,B 0,C 180,E1 -1626.591,E2 -1626.591} C_VEL
LIN {X 0,Y 587.276,Z 379.517,A -85,B 0,C 180,E1 -1627.737,E2 -1627.737} C_VEL
LIN {X 0,Y 587.337,Z 371.092,A -85,B 0,C 180,E1 -1628.776,E2 -1628.776} C_VEL
LIN {X 0,Y 587.419,Z 360.934,A -85,B 0,C 180,E1 -1629.817,E2 -1629.817} C_VEL
LIN {X 0,Y 587.524,Z 349.555,A -85,B 0,C 180,E1 -1630.773,E2 -1630.773} C_VEL
LIN {X 0,Y 587.634,Z 338.136,A -85,B 0,C 180,E1 -1631.565,E2 -1631.565} C_VEL
LIN {X 0,Y 587.727,Z 325.884,A -85,B 0,C 180,E1 -1632.255,E2 -1632.255} C_VEL
LIN {X 0,Y 587.837,Z 312.076,A -85,B 0,C 180,E1 -1632.866,E2 -1632.866} C_VEL
LIN {X 0,Y 587.658,Z 301.252,A -85,B 0,C 180,E1 -1633.244,E2 -1633.244} C_VEL
LIN {X 0,Y 587.393,Z 300.245,A -85,B 0,C 180,E1 -1633.34,E2 -1633.34} C_VEL
LIN {X 0,Y 586.867,Z 300.005,A -85,B 0,C 180,E1 -1633.693,E2 -1633.693} C_VEL
LIN {X 0,Y 583.579,Z 300.42,A -85,B 0,C 180,E1 -1634.799,E2 -1634.799} C_VEL
LIN {X 0,Y 581.305,Z 300.891,A -85,B 0,C 180,E1 -1635.566,E2 -1635.566} C_VEL
LIN {X 0,Y 580.354,Z 300.837,A -85,B 0,C 180,E1 -1636.159,E2 -1636.159} C_VEL
LIN {X 0,Y 580.282,Z 300.826,A -85,B 0,C 180,E1 -1636.359,E2 -1636.359} C_VEL
LIN {X 0,Y 580.327,Z 300.822,A -85,B 0,C 180,E1 -1639.158,E2 -1639.158} C_VEL
LIN {X 0,Y 580.277,Z 300.824,A -85,B 0,C 180,E1 -1642.053,E2 -1642.053} C_VEL
LIN {X 0,Y 580.31,Z 300.823,A -85,B 0,C 180,E1 -1645.08,E2 -1645.08} C_VEL
LIN {X 0,Y 580.304,Z 300.822,A -85,B 0,C 180,E1 -1648.186,E2 -1648.186} C_VEL
LIN {X 0,Y 580.289,Z 300.83,A -85,B 0,C 180,E1 -1650.695,E2 -1650.695} C_VEL
LIN {X 0,Y 580.307,Z 300.819,A -85,B 0,C 180,E1 -1653.316,E2 -1653.316} C_VEL
LIN {X 0,Y 580.282,Z 300.822,A -85,B 0,C 180,E1 -1655.761,E2 -1655.761} C_VEL
LIN {X 0,Y 580.293,Z 300.824,A -85,B 0,C 180,E1 -1658.146,E2 -1658.146} C_VEL
LIN {X 0,Y 580.303,Z 300.823,A -85,B 0,C 180,E1 -1660.844,E2 -1660.844} C_VEL
LIN {X 0,Y 580.284,Z 300.822,A -85,B 0,C 180,E1 -1663.658,E2 -1663.658} C_VEL
LIN {X 0,Y 580.291,Z 300.827,A -85,B 0,C 180,E1 -1666.608,E2 -1666.608} C_VEL
LIN {X 0,Y 580.303,Z 300.819,A -85,B 0,C 180,E1 -1669.157,E2 -1669.157} C_VEL
LIN {X 0,Y 580.294,Z 300.824,A -85,B 0,C 180,E1 -1671.927,E2 -1671.927} C_VEL
LIN {X 0,Y 580.258,Z 300.832,A -85,B 0,C 180,E1 -1674.453,E2 -1674.453} C_VEL
LIN {X 0,Y 580.298,Z 300.82,A -85,B 0,C 180,E1 -1676.975,E2 -1676.975} C_VEL
LIN {X 0,Y 580.301,Z 300.82,A -85,B 0,C 180,E1 -1679.425,E2 -1679.425} C_VEL
LIN {X 0,Y 580.306,Z 300.829,A -85,B 0,C 180,E1 -1682.141,E2 -1682.141} C_VEL
LIN {X 0,Y 580.328,Z 300.816,A -85,B 0,C 180,E1 -1685.27,E2 -1685.27} C_VEL
LIN {X 0,Y 580.279,Z 300.83,A -85,B 0,C 180,E1 -1687.947,E2 -1687.947} C_VEL
LIN {X 0,Y 580.304,Z 300.819,A -85,B 0,C 180,E1 -1690.913,E2 -1690.913} C_VEL
LIN {X 0,Y 580.317,Z 300.817,A -85,B 0,C 180,E1 -1693.102,E2 -1693.102} C_VEL
LIN {X 0,Y 580.332,Z 300.826,A -85,B 0,C 180,E1 -1695.983,E2 -1695.983} C_VEL
LIN {X 0,Y 580.312,Z 300.818,A -85,B 0,C 180,E1 -1698.826,E2 -1698.826} C_VEL
LIN {X 0,Y 580.334,Z 300.822,A -85,B 0,C 180,E1 -1701.643,E2 -1701.643} C_VEL
LIN {X 0,Y 580.331,Z 300.817,A -85,B 0,C 180,E1 -1704.44,E2 -1704.44} C_VEL
LIN {X 0,Y 580.347,Z 300.821,A -85,B 0,C 180,E1 -1707.917,E2 -1707.917} C_VEL
LIN {X 0,Y 580.363,Z 300.812,A -85,B 0,C 180,E1 -1710.693,E2 -1710.693} C_VEL
LIN {X 0,Y 580.287,Z 300.828,A -85,B 0,C 180,E1 -1713.471,E2 -1713.471} C_VEL
LIN {X 0,Y 580.328,Z 300.824,A -85,B 0,C 180,E1 -1715.559,E2 -1715.559} C_VEL
LIN {X 0,Y 580.332,Z 300.816,A -85,B 0,C 180,E1 -1718.355,E2 -1718.355} C_VEL
LIN {X 0,Y 580.305,Z 300.823,A -85,B 0,C 180,E1 -1721.19,E2 -1721.19} C_VEL
LIN {X 0,Y 580.33,Z 300.818,A -85,B 0,C 180,E1 -1724.016,E2 -1724.016} C_VEL
LIN {X 0,Y 580.316,Z 300.819,A -85,B 0,C 180,E1 -1726.913,E2 -1726.913} C_VEL
LIN {X 0,Y 580.307,Z 300.823,A -85,B 0,C 180,E1 -1729.821,E2 -1729.821} C_VEL
LIN {X 0,Y 580.298,Z 300.821,A -85,B 0,C 180,E1 -1732.801,E2 -1732.801} C_VEL
LIN {X 0,Y 580.309,Z 300.824,A -85,B 0,C 180,E1 -1735.079,E2 -1735.079} C_VEL
LIN {X 0,Y 580.301,Z 300.819,A -85,B 0,C 180,E1 -1738.185,E2 -1738.185} C_VEL
LIN {X 0,Y 580.292,Z 300.822,A -85,B 0,C 180,E1 -1740.695,E2 -1740.695} C_VEL
LIN {X 0,Y 580.305,Z 300.828,A -85,B 0,C 180,E1 -1743.316,E2 -1743.316} C_VEL
LIN {X 0,Y 580.248,Z 300.828,A -85,B 0,C 180,E1 -1745.756,E2 -1745.756} C_VEL
LIN {X 0,Y 580.288,Z 300.821,A -85,B 0,C 180,E1 -1748.145,E2 -1748.145} C_VEL
LIN {X 0,Y 580.299,Z 300.825,A -85,B 0,C 180,E1 -1750.842,E2 -1750.842} C_VEL
LIN {X 0,Y 580.286,Z 300.823,A -85,B 0,C 180,E1 -1753.656,E2 -1753.656} C_VEL
LIN {X 0,Y 580.282,Z 300.825,A -85,B 0,C 180,E1 -1756.607,E2 -1756.607} C_VEL
LIN {X 0,Y 580.298,Z 300.827,A -85,B 0,C 180,E1 -1759.156,E2 -1759.156} C_VEL
LIN {X 0,Y 580.288,Z 300.821,A -85,B 0,C 180,E1 -1761.926,E2 -1761.926} C_VEL
LIN {X 0,Y 580.304,Z 300.822,A -85,B 0,C 180,E1 -1764.456,E2 -1764.456} C_VEL
LIN {X 0,Y 580.286,Z 300.83,A -85,B 0,C 180,E1 -1766.975,E2 -1766.975} C_VEL
LIN {X 0,Y 580.306,Z 300.821,A -85,B 0,C 180,E1 -1769.425,E2 -1769.425} C_VEL
LIN {X 0,Y 580.314,Z 300.819,A -85,B 0,C 180,E1 -1772.136,E2 -1772.136} C_VEL
LIN {X 0,Y 580.303,Z 300.827,A -85,B 0,C 180,E1 -1774.92,E2 -1774.92} C_VEL
LIN {X 0,Y 580.27,Z 300.824,A -85,B 0,C 180,E1 -1777.947,E2 -1777.947} C_VEL
LIN {X 0,Y 580.312,Z 300.824,A -85,B 0,C 180,E1 -1780.914,E2 -1780.914} C_VEL
LIN {X 0,Y 580.278,Z 300.823,A -85,B 0,C 180,E1 -1783.825,E2 -1783.825} C_VEL
LIN {X 0,Y 580.321,Z 300.818,A -85,B 0,C 180,E1 -1785.983,E2 -1785.983} C_VEL
LIN {X 0,Y 580.296,Z 300.825,A -85,B 0,C 180,E1 -1788.826,E2 -1788.826} C_VEL
LIN {X 0,Y 580.328,Z 300.816,A -85,B 0,C 180,E1 -1791.644,E2 -1791.644} C_VEL
LIN {X 0,Y 580.322,Z 300.827,A -85,B 0,C 180,E1 -1794.44,E2 -1794.44} C_VEL
LIN {X 0,Y 580.339,Z 300.815,A -85,B 0,C 180,E1 -1797.223,E2 -1797.223} C_VEL
LIN {X 0,Y 580.345,Z 300.818,A -85,B 0,C 180,E1 -1800,E2 -1800} C_VEL
LIN {X 0,Y 580.338,Z 300.818,A -85,B 0,C 180,E1 -1802.776,E2 -1802.776} C_VEL
LIN {X 0,Y 580.32,Z 300.818,A -85,B 0,C 180,E1 -1805.56,E2 -1805.56} C_VEL
LIN {X 0,Y 580.328,Z 300.825,A -85,B 0,C 180,E1 -1808.356,E2 -1808.356} C_VEL
LIN {X 0,Y 580.291,Z 300.82,A -85,B 0,C 180,E1 -1811.191,E2 -1811.191} C_VEL
LIN {X 0,Y 580.32,Z 300.825,A -85,B 0,C 180,E1 -1814.017,E2 -1814.017} C_VEL
LIN {X 0,Y 580.306,Z 300.819,A -85,B 0,C 180,E1 -1816.915,E2 -1816.915} C_VEL
LIN {X 0,Y 580.301,Z 300.825,A -85,B 0,C 180,E1 -1819.822,E2 -1819.822} C_VEL
LIN {X 0,Y 580.288,Z 300.821,A -85,B 0,C 180,E1 -1822.803,E2 -1822.803} C_VEL
LIN {X 0,Y 580.3,Z 300.819,A -85,B 0,C 180,E1 -1825.08,E2 -1825.08} C_VEL
LIN {X 0,Y 580.295,Z 300.826,A -85,B 0,C 180,E1 -1828.186,E2 -1828.186} C_VEL
LIN {X 0,Y 580.293,Z 300.821,A -85,B 0,C 180,E1 -1830.698,E2 -1830.698} C_VEL
LIN {X 0,Y 580.297,Z 300.822,A -85,B 0,C 180,E1 -1833.317,E2 -1833.317} C_VEL
LIN {X 0,Y 580.321,Z 300.826,A -85,B 0,C 180,E1 -1835.768,E2 -1835.768} C_VEL
LIN {X 0,Y 580.284,Z 300.827,A -85,B 0,C 180,E1 -1838.147,E2 -1838.147} C_VEL
LIN {X 0,Y 580.295,Z 300.821,A -85,B 0,C 180,E1 -1840.844,E2 -1840.844} C_VEL
LIN {X 0,Y 580.273,Z 300.833,A -85,B 0,C 180,E1 -1843.658,E2 -1843.658} C_VEL
LIN {X 0,Y 580.288,Z 300.823,A -85,B 0,C 180,E1 -1846.608,E2 -1846.608} C_VEL
LIN {X 0,Y 580.296,Z 300.827,A -85,B 0,C 180,E1 -1849.158,E2 -1849.158} C_VEL
LIN {X 0,Y 580.337,Z 301.035,A -85,B 0,C 180,E1 -1850.438,E2 -1850.438} C_VEL
LIN {X 0,Y 581.175,Z 305.383,A -85,B 0,C 180,E1 -1851.468,E2 -1851.468} C_VEL
LIN {X 0,Y 581.104,Z 315.45,A -85,B 0,C 180,E1 -1853.658,E2 -1853.658} C_VEL
LIN {X 0,Y 580.944,Z 327.53,A -85,B 0,C 180,E1 -1856.188,E2 -1856.188} C_VEL
LIN {X 0,Y 580.937,Z 341.21,A -85,B 0,C 180,E1 -1858.97,E2 -1858.97} C_VEL
LIN {X 0,Y 580.916,Z 355.969,A -85,B 0,C 180,E1 -1861.848,E2 -1861.848} C_VEL
LIN {X 0,Y 580.785,Z 369.497,A -85,B 0,C 180,E1 -1864.56,E2 -1864.56} C_VEL
LIN {X 0,Y 580.638,Z 384.796,A -85,B 0,C 180,E1 -1867.588,E2 -1867.588} C_VEL
LIN {X 0,Y 580.493,Z 400.032,A -85,B 0,C 180,E1 -1870.541,E2 -1870.541} C_VEL
LIN {X 0,Y 580.377,Z 415.396,A -85,B 0,C 180,E1 -1873.468,E2 -1873.468} C_VEL
LIN {X 0,Y 580.361,Z 423.864,A -85,B 0,C 180,E1 -1875.022,E2 -1875.022} C_VEL
LIN {X 0,Y 581.09,Z 428.086,A -85,B 0,C 180,E1 -1875.129,E2 -1875.129} C_VEL
LIN {X 0,Y 581.075,Z 442.879,A -85,B 0,C 180,E1 -1875.41,E2 -1875.41} C_VEL
LIN {X 0,Y 580.992,Z 456.929,A -85,B 0,C 180,E1 -1875.823,E2 -1875.823} C_VEL
LIN {X 0,Y 580.868,Z 470.15,A -85,B 0,C 180,E1 -1876.354,E2 -1876.354} C_VEL
LIN {X 0,Y 580.703,Z 482.227,A -85,B 0,C 180,E1 -1876.974,E2 -1876.974} C_VEL
LIN {X 0,Y 580.588,Z 494.719,A -85,B 0,C 180,E1 -1877.771,E2 -1877.771} C_VEL
LIN {X 0,Y 580.465,Z 506.02,A -85,B 0,C 180,E1 -1878.654,E2 -1878.654} C_VEL
LIN {X 0,Y 580.356,Z 515.398,A -85,B 0,C 180,E1 -1879.535,E2 -1879.535} C_VEL
LIN {X 0,Y 580.286,Z 524.829,A -85,B 0,C 180,E1 -1880.59,E2 -1880.59} C_VEL
LIN {X 0,Y 580.192,Z 533.804,A -85,B 0,C 180,E1 -1881.818,E2 -1881.818} C_VEL
LIN {X 0,Y 580.14,Z 541.056,A -85,B 0,C 180,E1 -1883.043,E2 -1883.043} C_VEL
LIN {X 0,Y 580.128,Z 547.571,A -85,B 0,C 180,E1 -1884.439,E2 -1884.439} C_VEL
LIN {X 0,Y 580.102,Z 552.444,A -85,B 0,C 180,E1 -1885.832,E2 -1885.832} C_VEL
LIN {X 0,Y 580.041,Z 555.833,A -85,B 0,C 180,E1 -1887.223,E2 -1887.223} C_VEL
LIN {X 0,Y 580.041,Z 557.833,A -85,B 0,C 180,E1 -1888.612,E2 -1888.612} C_VEL
LIN {X 0,Y 580.036,Z 558.5,A -85,B 0,C 180,E1 -1890.001,E2 -1890.001} C_VEL
LIN {X 0,Y 580.041,Z 557.832,A -85,B 0,C 180,E1 -1891.389,E2 -1891.389} C_VEL
LIN {X 0,Y 580.041,Z 555.831,A -85,B 0,C 180,E1 -1892.779,E2 -1892.779} C_VEL
LIN {X 0,Y 580.102,Z 552.442,A -85,B 0,C 180,E1 -1894.169,E2 -1894.169} C_VEL
LIN {X 0,Y 580.128,Z 547.565,A -85,B 0,C 180,E1 -1895.562,E2 -1895.562} C_VEL
LIN {X 0,Y 580.141,Z 541.049,A -85,B 0,C 180,E1 -1896.959,E2 -1896.959} C_VEL
LIN {X 0,Y 580.192,Z 533.796,A -85,B 0,C 180,E1 -1898.183,E2 -1898.183} C_VEL
LIN {X 0,Y 580.284,Z 524.818,A -85,B 0,C 180,E1 -1899.411,E2 -1899.411} C_VEL
LIN {X 0,Y 580.356,Z 515.385,A -85,B 0,C 180,E1 -1900.466,E2 -1900.466} C_VEL
LIN {X 0,Y 580.476,Z 505.311,A -85,B 0,C 180,E1 -1901.405,E2 -1901.405} C_VEL
LIN {X 0,Y 580.596,Z 493.423,A -85,B 0,C 180,E1 -1902.319,E2 -1902.319} C_VEL
LIN {X 0,Y 580.731,Z 480.638,A -85,B 0,C 180,E1 -1903.116,E2 -1903.116} C_VEL
LIN {X 0,Y 580.868,Z 468.146,A -85,B 0,C 180,E1 -1903.736,E2 -1903.736} C_VEL
LIN {X 0,Y 580.999,Z 455.231,A -85,B 0,C 180,E1 -1904.235,E2 -1904.235} C_VEL
LIN {X 0,Y 581.083,Z 441.172,A -85,B 0,C 180,E1 -1904.631,E2 -1904.631} C_VEL
LIN {X 0,Y 581.088,Z 428.083,A -85,B 0,C 180,E1 -1904.871,E2 -1904.871} C_VEL
LIN {X 0,Y 580.377,Z 424.184,A -85,B 0,C 180,E1 -1904.957,E2 -1904.957} C_VEL
LIN {X 0,Y 580.342,Z 423.05,A -85,B 0,C 180,E1 -1905.092,E2 -1905.092} C_VEL
LIN {X 0,Y 580.402,Z 407.739,A -85,B 0,C 180,E1 -1907.986,E2 -1907.986} C_VEL
LIN {X 0,Y 580.553,Z 394.352,A -85,B 0,C 180,E1 -1910.553,E2 -1910.553} C_VEL
LIN {X 0,Y 580.684,Z 380.44,A -85,B 0,C 180,E1 -1913.267,E2 -1913.267} C_VEL
LIN {X 0,Y 580.829,Z 366.052,A -85,B 0,C 180,E1 -1916.131,E2 -1916.131} C_VEL
LIN {X 0,Y 580.886,Z 355.909,A -85,B 0,C 180,E1 -1918.155,E2 -1918.155} C_VEL
LIN {X 0,Y 580.747,Z 341.015,A -85,B 0,C 180,E1 -1920.771,E2 -1920.771} C_VEL
LIN {X 0,Y 580.402,Z 323.822,A -85,B 0,C 180,E1 -1923.85,E2 -1923.85} C_VEL
LIN {X 0,Y 580.567,Z 308.633,A -85,B 0,C 180,E1 -1926.677,E2 -1926.677} C_VEL
LIN {X 0,Y 580.572,Z 302.555,A -85,B 0,C 180,E1 -1927.869,E2 -1927.869} C_VEL
LIN {X 0,Y 580.316,Z 300.915,A -85,B 0,C 180,E1 -1928.255,E2 -1928.255} C_VEL
LIN {X 0,Y 580.303,Z 300.822,A -85,B 0,C 180,E1 -1930.844,E2 -1930.844} C_VEL
LIN {X 0,Y 580.292,Z 300.831,A -85,B 0,C 180,E1 -1933.657,E2 -1933.657} C_VEL
LIN {X 0,Y 580.28,Z 300.823,A -85,B 0,C 180,E1 -1936.61,E2 -1936.61} C_VEL
LIN {X 0,Y 580.303,Z 300.824,A -85,B 0,C 180,E1 -1939.157,E2 -1939.157} C_VEL
LIN {X 0,Y 580.294,Z 300.825,A -85,B 0,C 180,E1 -1941.927,E2 -1941.927} C_VEL
LIN {X 0,Y 580.309,Z 300.819,A -85,B 0,C 180,E1 -1944.457,E2 -1944.457} C_VEL
LIN {X 0,Y 580.294,Z 300.824,A -85,B 0,C 180,E1 -1946.975,E2 -1946.975} C_VEL
LIN {X 0,Y 580.299,Z 300.83,A -85,B 0,C 180,E1 -1949.425,E2 -1949.425} C_VEL
LIN {X 0,Y 580.324,Z 300.818,A -85,B 0,C 180,E1 -1952.137,E2 -1952.137} C_VEL
LIN {X 0,Y 580.325,Z 300.827,A -85,B 0,C 180,E1 -1955.27,E2 -1955.27} C_VEL
LIN {X 0,Y 580.276,Z 300.825,A -85,B 0,C 180,E1 -1957.948,E2 -1957.948} C_VEL
LIN {X 0,Y 580.323,Z 300.823,A -85,B 0,C 180,E1 -1960.914,E2 -1960.914} C_VEL
LIN {X 0,Y 580.283,Z 300.827,A -85,B 0,C 180,E1 -1963.826,E2 -1963.826} C_VEL
LIN {X 0,Y 580.328,Z 300.948,A -85,B 0,C 180,E1 -1964.548,E2 -1964.548} C_VEL
LIN {X 0,Y 580.455,Z 301.589,A -85,B 0,C 180,E1 -1964.664,E2 -1964.664} C_VEL
LIN {X 0,Y 580.971,Z 303.994,A -85,B 0,C 180,E1 -1964.768,E2 -1964.768} C_VEL
LIN {X 0,Y 580.906,Z 317.553,A -85,B 0,C 180,E1 -1965.282,E2 -1965.282} C_VEL
LIN {X 0,Y 580.768,Z 329.923,A -85,B 0,C 180,E1 -1965.89,E2 -1965.89} C_VEL
LIN {X 0,Y 580.632,Z 341.828,A -85,B 0,C 180,E1 -1966.615,E2 -1966.615} C_VEL
LIN {X 0,Y 580.497,Z 353.663,A -85,B 0,C 180,E1 -1967.502,E2 -1967.502} C_VEL
LIN {X 0,Y 580.381,Z 364.352,A -85,B 0,C 180,E1 -1968.475,E2 -1968.475} C_VEL
LIN {X 0,Y 580.323,Z 373.982,A -85,B 0,C 180,E1 -1969.534,E2 -1969.534} C_VEL
LIN {X 0,Y 580.21,Z 383.15,A -85,B 0,C 180,E1 -1970.764,E2 -1970.764} C_VEL
LIN {X 0,Y 580.154,Z 390.566,A -85,B 0,C 180,E1 -1971.992,E2 -1971.992} C_VEL
LIN {X 0,Y 580.139,Z 395.722,A -85,B 0,C 180,E1 -1973.042,E2 -1973.042} C_VEL
LIN {X 0,Y 580.117,Z 401.096,A -85,B 0,C 180,E1 -1974.438,E2 -1974.438} C_VEL
LIN {X 0,Y 580.087,Z 404.924,A -85,B 0,C 180,E1 -1975.832,E2 -1975.832} C_VEL
LIN {X 0,Y 580.04,Z 407.354,A -85,B 0,C 180,E1 -1977.222,E2 -1977.222} C_VEL
LIN {X 0,Y 580.046,Z 408.418,A -85,B 0,C 180,E1 -1978.612,E2 -1978.612} C_VEL
LIN {X 0,Y 580.036,Z 408.166,A -85,B 0,C 180,E1 -1980,E2 -1980} C_VEL
LIN {X 0,Y 580.048,Z 406.618,A -85,B 0,C 180,E1 -1981.389,E2 -1981.389} C_VEL
LIN {X 0,Y 580.048,Z 403.669,A -85,B 0,C 180,E1 -1982.778,E2 -1982.778} C_VEL
LIN {X 0,Y 580.106,Z 399.286,A -85,B 0,C 180,E1 -1984.169,E2 -1984.169} C_VEL
LIN {X 0,Y 580.137,Z 393.325,A -85,B 0,C 180,E1 -1985.562,E2 -1985.562} C_VEL
LIN {X 0,Y 580.15,Z 386.687,A -85,B 0,C 180,E1 -1986.773,E2 -1986.773} C_VEL
LIN {X 0,Y 580.242,Z 378.313,A -85,B 0,C 180,E1 -1988.007,E2 -1988.007} C_VEL
LIN {X 0,Y 580.315,Z 369.66,A -85,B 0,C 180,E1 -1989.058,E2 -1989.058} C_VEL
LIN {X 0,Y 580.452,Z 359.141,A -85,B 0,C 180,E1 -1990.112,E2 -1990.112} C_VEL
LIN {X 0,Y 580.573,Z 347.418,A -85,B 0,C 180,E1 -1991.08,E2 -1991.08} C_VEL
LIN {X 0,Y 580.71,Z 335.589,A -85,B 0,C 180,E1 -1991.873,E2 -1991.873} C_VEL
LIN {X 0,Y 580.873,Z 322.564,A -85,B 0,C 180,E1 -1992.579,E2 -1992.579} C_VEL
LIN {X 0,Y 580.986,Z 308.877,A -85,B 0,C 180,E1 -1993.154,E2 -1993.154} C_VEL
LIN {X 0,Y 580.975,Z 303.648,A -85,B 0,C 180,E1 -1993.332,E2 -1993.332} C_VEL
LIN {X 0,Y 580.391,Z 301.292,A -85,B 0,C 180,E1 -1993.458,E2 -1993.458} C_VEL
LIN {X 0,Y 580.329,Z 300.834,A -85,B 0,C 180,E1 -1993.66,E2 -1993.66} C_VEL
LIN {X 0,Y 580.282,Z 300.826,A -85,B 0,C 180,E1 -1996.359,E2 -1996.359} C_VEL
LIN {X 0,Y 579.638,Z 300.911,A -85,B 0,C 180,E1 -1996.938,E2 -1996.938} C_VEL
LIN {X 0,Y 576.82,Z 301.263,A -85,B 0,C 180,E1 -1997.878,E2 -1997.878} C_VEL
LIN {X 0,Y 574.418,Z 301.561,A -85,B 0,C 180,E1 -1998.634,E2 -1998.634} C_VEL
LIN {X 0,Y 573.367,Z 301.689,A -85,B 0,C 180,E1 -1999.217,E2 -1999.217} C_VEL
LIN {X 0,Y 573.272,Z 301.698,A -85,B 0,C 180,E1 -1999.415,E2 -1999.415} C_VEL
LIN {X 0,Y 573.241,Z 301.703,A -85,B 0,C 180,E1 -2002.338,E2 -2002.338} C_VEL
LIN {X 0,Y 573.257,Z 301.698,A -85,B 0,C 180,E1 -2005.41,E2 -2005.41} C_VEL
LIN {X 0,Y 573.256,Z 301.698,A -85,B 0,C 180,E1 -2008.029,E2 -2008.029} C_VEL
LIN {X 0,Y 573.251,Z 301.7,A -85,B 0,C 180,E1 -2010.176,E2 -2010.176} C_VEL
LIN {X 0,Y 573.258,Z 301.706,A -85,B 0,C 180,E1 -2012.645,E2 -2012.645} C_VEL
LIN {X 0,Y 573.26,Z 301.698,A -85,B 0,C 180,E1 -2015.185,E2 -2015.185} C_VEL
LIN {X 0,Y 573.241,Z 301.7,A -85,B 0,C 180,E1 -2017.808,E2 -2017.808} C_VEL
LIN {X 0,Y 573.25,Z 301.708,A -85,B 0,C 180,E1 -2020.525,E2 -2020.525} C_VEL
LIN {X 0,Y 573.244,Z 301.698,A -85,B 0,C 180,E1 -2023.359,E2 -2023.359} C_VEL
LIN {X 0,Y 573.259,Z 301.706,A -85,B 0,C 180,E1 -2026.33,E2 -2026.33} C_VEL
LIN {X 0,Y 573.25,Z 301.705,A -85,B 0,C 180,E1 -2028.544,E2 -2028.544} C_VEL
LIN {X 0,Y 573.245,Z 301.698,A -85,B 0,C 180,E1 -2031.298,E2 -2031.298} C_VEL
LIN {X 0,Y 573.219,Z 301.707,A -85,B 0,C 180,E1 -2034.018,E2 -2034.018} C_VEL
LIN {X 0,Y 573.276,Z 301.7,A -85,B 0,C 180,E1 -2036.518,E2 -2036.518} C_VEL
LIN {X 0,Y 573.234,Z 301.7,A -85,B 0,C 180,E1 -2039.118,E2 -2039.118} C_VEL
LIN {X 0,Y 573.245,Z 301.699,A -85,B 0,C 180,E1 -2041.435,E2 -2041.435} C_VEL
LIN {X 0,Y 573.272,Z 301.7,A -85,B 0,C 180,E1 -2043.81,E2 -2043.81} C_VEL
LIN {X 0,Y 573.234,Z 301.71,A -85,B 0,C 180,E1 -2046.134,E2 -2046.134} C_VEL
LIN {X 0,Y 573.257,Z 301.697,A -85,B 0,C 180,E1 -2049.173,E2 -2049.173} C_VEL
LIN {X 0,Y 573.235,Z 301.701,A -85,B 0,C 180,E1 -2051.411,E2 -2051.411} C_VEL
LIN {X 0,Y 573.257,Z 301.701,A -85,B 0,C 180,E1 -2053.621,E2 -2053.621} C_VEL
LIN {X 0,Y 573.28,Z 301.702,A -85,B 0,C 180,E1 -2055.807,E2 -2055.807} C_VEL
LIN {X 0,Y 573.27,Z 301.695,A -85,B 0,C 180,E1 -2058.745,E2 -2058.745} C_VEL
LIN {X 0,Y 573.29,Z 301.697,A -85,B 0,C 180,E1 -2061.54,E2 -2061.54} C_VEL
LIN {X 0,Y 573.299,Z 301.694,A -85,B 0,C 180,E1 -2064.371,E2 -2064.371} C_VEL
LIN {X 0,Y 573.318,Z 301.697,A -85,B 0,C 180,E1 -2067.892,E2 -2067.892} C_VEL
LIN {X 0,Y 573.334,Z 301.687,A -85,B 0,C 180,E1 -2070.702,E2 -2070.702} C_VEL
LIN {X 0,Y 573.307,Z 301.691,A -85,B 0,C 180,E1 -2072.81,E2 -2072.81} C_VEL
LIN {X 0,Y 573.296,Z 301.702,A -85,B 0,C 180,E1 -2075.627,E2 -2075.627} C_VEL
LIN {X 0,Y 573.288,Z 301.693,A -85,B 0,C 180,E1 -2078.459,E2 -2078.459} C_VEL
LIN {X 0,Y 573.277,Z 301.7,A -85,B 0,C 180,E1 -2081.311,E2 -2081.311} C_VEL
LIN {X 0,Y 573.286,Z 301.693,A -85,B 0,C 180,E1 -2084.424,E2 -2084.424} C_VEL
LIN {X 0,Y 573.262,Z 301.7,A -85,B 0,C 180,E1 -2087.111,E2 -2087.111} C_VEL
LIN {X 0,Y 573.254,Z 301.699,A -85,B 0,C 180,E1 -2090.076,E2 -2090.076} C_VEL
LIN {X 0,Y 573.237,Z 301.705,A -85,B 0,C 180,E1 -2093.098,E2 -2093.098} C_VEL
LIN {X 0,Y 573.257,Z 301.706,A -85,B 0,C 180,E1 -2095.409,E2 -2095.409} C_VEL
LIN {X 0,Y 573.253,Z 301.698,A -85,B 0,C 180,E1 -2098.028,E2 -2098.028} C_VEL
LIN {X 0,Y 573.239,Z 301.703,A -85,B 0,C 180,E1 -2100.883,E2 -2100.883} C_VEL
LIN {X 0,Y 573.262,Z 301.702,A -85,B 0,C 180,E1 -2103.523,E2 -2103.523} C_VEL
LIN {X 0,Y 573.215,Z 301.702,A -85,B 0,C 180,E1 -2106.05,E2 -2106.05} C_VEL
LIN {X 0,Y 573.248,Z 301.701,A -85,B 0,C 180,E1 -2108.7,E2 -2108.7} C_VEL
LIN {X 0,Y 573.252,Z 301.7,A -85,B 0,C 180,E1 -2111.595,E2 -2111.595} C_VEL
LIN {X 0,Y 573.237,Z 301.7,A -85,B 0,C 180,E1 -2114.332,E2 -2114.332} C_VEL
LIN {X 0,Y 573.24,Z 301.704,A -85,B 0,C 180,E1 -2117.357,E2 -2117.357} C_VEL
LIN {X 0,Y 573.246,Z 301.7,A -85,B 0,C 180,E1 -2120.392,E2 -2120.392} C_VEL
LIN {X 0,Y 573.253,Z 301.705,A -85,B 0,C 180,E1 -2123.077,E2 -2123.077} C_VEL
LIN {X 0,Y 573.27,Z 301.696,A -85,B 0,C 180,E1 -2125.671,E2 -2125.671} C_VEL
LIN {X 0,Y 573.245,Z 301.699,A -85,B 0,C 180,E1 -2128.184,E2 -2128.184} C_VEL
LIN {X 0,Y 573.264,Z 301.703,A -85,B 0,C 180,E1 -2130.634,E2 -2130.634} C_VEL
LIN {X 0,Y 573.266,Z 301.696,A -85,B 0,C 180,E1 -2133.5,E2 -2133.5} C_VEL
LIN {X 0,Y 573.228,Z 301.702,A -85,B 0,C 180,E1 -2136.134,E2 -2136.134} C_VEL
LIN {X 0,Y 573.245,Z 301.701,A -85,B 0,C 180,E1 -2139.173,E2 -2139.173} C_VEL
LIN {X 0,Y 573.232,Z 301.701,A -85,B 0,C 180,E1 -2141.411,E2 -2141.411} C_VEL
LIN {X 0,Y 573.253,Z 301.697,A -85,B 0,C 180,E1 -2143.622,E2 -2143.622} C_VEL
LIN {X 0,Y 573.234,Z 301.709,A -85,B 0,C 180,E1 -2146.529,E2 -2146.529} C_VEL
LIN {X 0,Y 573.255,Z 301.704,A -85,B 0,C 180,E1 -2148.745,E2 -2148.745} C_VEL
LIN {X 0,Y 573.284,Z 301.693,A -85,B 0,C 180,E1 -2151.54,E2 -2151.54} C_VEL
LIN {X 0,Y 573.288,Z 301.702,A -85,B 0,C 180,E1 -2154.372,E2 -2154.372} C_VEL
LIN {X 0,Y 573.304,Z 301.693,A -85,B 0,C 180,E1 -2157.892,E2 -2157.892} C_VEL
LIN {X 0,Y 573.329,Z 301.692,A -85,B 0,C 180,E1 -2160.702,E2 -2160.702} C_VEL
LIN {X 0,Y 573.233,Z 301.7,A -85,B 0,C 180,E1 -2163.514,E2 -2163.514} C_VEL
LIN {X 0,Y 573.287,Z 301.694,A -85,B 0,C 180,E1 -2165.628,E2 -2165.628} C_VEL
LIN {X 0,Y 573.284,Z 301.7,A -85,B 0,C 180,E1 -2168.459,E2 -2168.459} C_VEL
LIN {X 0,Y 573.263,Z 301.696,A -85,B 0,C 180,E1 -2171.312,E2 -2171.312} C_VEL
LIN {X 0,Y 573.267,Z 301.706,A -85,B 0,C 180,E1 -2174.193,E2 -2174.193} C_VEL
LIN {X 0,Y 573.252,Z 301.697,A -85,B 0,C 180,E1 -2177.112,E2 -2177.112} C_VEL
LIN {X 0,Y 573.247,Z 301.708,A -85,B 0,C 180,E1 -2180.077,E2 -2180.077} C_VEL
LIN {X 0,Y 573.226,Z 301.701,A -85,B 0,C 180,E1 -2183.1,E2 -2183.1} C_VEL
LIN {X 0,Y 573.248,Z 301.7,A -85,B 0,C 180,E1 -2185.41,E2 -2185.41} C_VEL
LIN {X 0,Y 573.257,Z 301.706,A -85,B 0,C 180,E1 -2188.032,E2 -2188.032} C_VEL
LIN {X 0,Y 573.237,Z 301.699,A -85,B 0,C 180,E1 -2190.885,E2 -2190.885} C_VEL
LIN {X 0,Y 573.255,Z 301.701,A -85,B 0,C 180,E1 -2193.524,E2 -2193.524} C_VEL
LIN {X 0,Y 573.255,Z 301.704,A -85,B 0,C 180,E1 -2196.049,E2 -2196.049} C_VEL
LIN {X 0,Y 573.244,Z 301.699,A -85,B 0,C 180,E1 -2198.701,E2 -2198.701} C_VEL
LIN {X 0,Y 573.248,Z 301.706,A -85,B 0,C 180,E1 -2201.596,E2 -2201.596} C_VEL
LIN {X 0,Y 573.23,Z 301.704,A -85,B 0,C 180,E1 -2204.334,E2 -2204.334} C_VEL
LIN {X 0,Y 573.246,Z 301.706,A -85,B 0,C 180,E1 -2207.358,E2 -2207.358} C_VEL
LIN {X 0,Y 573.275,Z 301.87,A -85,B 0,C 180,E1 -2210.14,E2 -2210.14} C_VEL
LIN {X 0,Y 574.35,Z 307.754,A -85,B 0,C 180,E1 -2211.548,E2 -2211.548} C_VEL
LIN {X 0,Y 574.202,Z 319.016,A -85,B 0,C 180,E1 -2214.021,E2 -2214.021} C_VEL
LIN {X 0,Y 574.006,Z 334.116,A -85,B 0,C 180,E1 -2217.196,E2 -2217.196} C_VEL
LIN {X 0,Y 573.961,Z 347.28,A -85,B 0,C 180,E1 -2219.866,E2 -2219.866} C_VEL
LIN {X 0,Y 573.922,Z 361.551,A -85,B 0,C 180,E1 -2222.665,E2 -2222.665} C_VEL
LIN {X 0,Y 573.825,Z 373.305,A -85,B 0,C 180,E1 -2225.002,E2 -2225.002} C_VEL
LIN {X 0,Y 573.645,Z 386.709,A -85,B 0,C 180,E1 -2227.68,E2 -2227.68} C_VEL
LIN {X 0,Y 573.496,Z 402.009,A -85,B 0,C 180,E1 -2230.679,E2 -2230.679} C_VEL
LIN {X 0,Y 573.326,Z 417.309,A -85,B 0,C 180,E1 -2233.625,E2 -2233.625} C_VEL
LIN {X 0,Y 573.335,Z 423.864,A -85,B 0,C 180,E1 -2234.834,E2 -2234.834} C_VEL
LIN {X 0,Y 573.994,Z 427.793,A -85,B 0,C 180,E1 -2234.937,E2 -2234.937} C_VEL
LIN {X 0,Y 574.291,Z 432.684,A -85,B 0,C 180,E1 -2235.018,E2 -2235.018} C_VEL
LIN {X 0,Y 574.172,Z 447.139,A -85,B 0,C 180,E1 -2235.34,E2 -2235.34} C_VEL
LIN {X 0,Y 574.015,Z 461.73,A -85,B 0,C 180,E1 -2235.827,E2 -2235.827} C_VEL
LIN {X 0,Y 573.869,Z 475.656,A -85,B 0,C 180,E1 -2236.455,E2 -2236.455} C_VEL
LIN {X 0,Y 573.72,Z 488.111,A -85,B 0,C 180,E1 -2237.173,E2 -2237.173} C_VEL
LIN {X 0,Y 573.533,Z 500.65,A -85,B 0,C 180,E1 -2238.067,E2 -2238.067} C_VEL
LIN {X 0,Y 573.436,Z 512.186,A -85,B 0,C 180,E1 -2239.084,E2 -2239.084} C_VEL
LIN {X 0,Y 573.239,Z 521.857,A -85,B 0,C 180,E1 -2240.117,E2 -2240.117} C_VEL
LIN {X 0,Y 573.202,Z 530.177,A -85,B 0,C 180,E1 -2241.185,E2 -2241.185} C_VEL
LIN {X 0,Y 573.109,Z 538.13,A -85,B 0,C 180,E1 -2242.426,E2 -2242.426} C_VEL
LIN {X 0,Y 573.021,Z 544.531,A -85,B 0,C 180,E1 -2243.663,E2 -2243.663} C_VEL
LIN {X 0,Y 573.001,Z 548.964,A -85,B 0,C 180,E1 -2244.723,E2 -2244.723} C_VEL
LIN {X 0,Y 573.028,Z 552.445,A -85,B 0,C 180,E1 -2245.781,E2 -2245.781} C_VEL
LIN {X 0,Y 572.956,Z 555.833,A -85,B 0,C 180,E1 -2247.188,E2 -2247.188} C_VEL
LIN {X 0,Y 572.941,Z 557.833,A -85,B 0,C 180,E1 -2248.595,E2 -2248.595} C_VEL
LIN {X 0,Y 572.937,Z 558.5,A -85,B 0,C 180,E1 -2250.001,E2 -2250.001} C_VEL
LIN {X 0,Y 572.941,Z 557.832,A -85,B 0,C 180,E1 -2251.406,E2 -2251.406} C_VEL
LIN {X 0,Y 572.956,Z 555.832,A -85,B 0,C 180,E1 -2252.813,E2 -2252.813} C_VEL
LIN {X 0,Y 573.028,Z 552.442,A -85,B 0,C 180,E1 -2254.221,E2 -2254.221} C_VEL
LIN {X 0,Y 573.057,Z 547.565,A -85,B 0,C 180,E1 -2255.631,E2 -2255.631} C_VEL
LIN {X 0,Y 573.065,Z 542.816,A -85,B 0,C 180,E1 -2256.7,E2 -2256.7} C_VEL
LIN {X 0,Y 573.126,Z 536.034,A -85,B 0,C 180,E1 -2257.93,E2 -2257.93} C_VEL
LIN {X 0,Y 573.226,Z 527.555,A -85,B 0,C 180,E1 -2259.172,E2 -2259.172} C_VEL
LIN {X 0,Y 573.304,Z 518.702,A -85,B 0,C 180,E1 -2260.239,E2 -2260.239} C_VEL
LIN {X 0,Y 573.463,Z 507.985,A -85,B 0,C 180,E1 -2261.309,E2 -2261.309} C_VEL
LIN {X 0,Y 573.59,Z 497.136,A -85,B 0,C 180,E1 -2262.203,E2 -2262.203} C_VEL
LIN {X 0,Y 573.767,Z 485.25,A -85,B 0,C 180,E1 -2263.008,E2 -2263.008} C_VEL
LIN {X 0,Y 573.952,Z 472.083,A -85,B 0,C 180,E1 -2263.725,E2 -2263.725} C_VEL
LIN {X 0,Y 574.094,Z 458.814,A -85,B 0,C 180,E1 -2264.284,E2 -2264.284} C_VEL
LIN {X 0,Y 574.201,Z 444.807,A -85,B 0,C 180,E1 -2264.72,E2 -2264.72} C_VEL
LIN {X 0,Y 574.291,Z 431.095,A -85,B 0,C 180,E1 -2265.006,E2 -2265.006} C_VEL
LIN {X 0,Y 573.795,Z 426.562,A -85,B 0,C 180,E1 -2265.087,E2 -2265.087} C_VEL
LIN {X 0,Y 573.336,Z 423.846,A -85,B 0,C 180,E1 -2265.168,E2 -2265.168} C_VEL
LIN {X 0,Y 573.392,Z 409.652,A -85,B 0,C 180,E1 -2267.844,E2 -2267.844} C_VEL
LIN {X 0,Y 573.528,Z 396.264,A -85,B 0,C 180,E1 -2270.441,E2 -2270.441} C_VEL
LIN {X 0,Y 573.723,Z 380.78,A -85,B 0,C 180,E1 -2273.498,E2 -2273.498} C_VEL
LIN {X 0,Y 573.895,Z 367.577,A -85,B 0,C 180,E1 -2276.159,E2 -2276.159} C_VEL
LIN {X 0,Y 573.842,Z 357.857,A -85,B 0,C 180,E1 -2277.935,E2 -2277.935} C_VEL
LIN {X 0,Y 573.697,Z 343.1,A -85,B 0,C 180,E1 -2280.552,E2 -2280.552} C_VEL
LIN {X 0,Y 573.363,Z 326.976,A -85,B 0,C 180,E1 -2283.476,E2 -2283.476} C_VEL
LIN {X 0,Y 573.542,Z 312.268,A -85,B 0,C 180,E1 -2286.245,E2 -2286.245} C_VEL
LIN {X 0,Y 573.688,Z 304.55,A -85,B 0,C 180,E1 -2287.773,E2 -2287.773} C_VEL
LIN {X 0,Y 573.28,Z 301.795,A -85,B 0,C 180,E1 -2288.395,E2 -2288.395} C_VEL
LIN {X 0,Y 573.248,Z 301.707,A -85,B 0,C 180,E1 -2291.456,E2 -2291.456} C_VEL
LIN {X 0,Y 573.243,Z 301.701,A -85,B 0,C 180,E1 -2294.333,E2 -2294.333} C_VEL
LIN {X 0,Y 573.244,Z 301.707,A -85,B 0,C 180,E1 -2297.359,E2 -2297.359} C_VEL
LIN {X 0,Y 573.251,Z 301.699,A -85,B 0,C 180,E1 -2300.393,E2 -2300.393} C_VEL
LIN {X 0,Y 573.26,Z 301.701,A -85,B 0,C 180,E1 -2303.078,E2 -2303.078} C_VEL
LIN {X 0,Y 573.277,Z 301.702,A -85,B 0,C 180,E1 -2305.672,E2 -2305.672} C_VEL
LIN {X 0,Y 573.244,Z 301.7,A -85,B 0,C 180,E1 -2308.185,E2 -2308.185} C_VEL
LIN {X 0,Y 573.268,Z 301.697,A -85,B 0,C 180,E1 -2310.634,E2 -2310.634} C_VEL
LIN {X 0,Y 573.254,Z 301.703,A -85,B 0,C 180,E1 -2313.024,E2 -2313.024} C_VEL
LIN {X 0,Y 573.278,Z 301.704,A -85,B 0,C 180,E1 -2315.366,E2 -2315.366} C_VEL
LIN {X 0,Y 573.232,Z 301.702,A -85,B 0,C 180,E1 -2318.42,E2 -2318.42} C_VEL
LIN {X 0,Y 573.282,Z 301.698,A -85,B 0,C 180,E1 -2320.728,E2 -2320.728} C_VEL
LIN {X 0,Y 573.255,Z 301.705,A -85,B 0,C 180,E1 -2323.622,E2 -2323.622} C_VEL
LIN {X 0,Y 573.335,Z 301.995,A -85,B 0,C 180,E1 -2324.446,E2 -2324.446} C_VEL
LIN {X 0,Y 573.538,Z 302.937,A -85,B 0,C 180,E1 -2324.543,E2 -2324.543} C_VEL
LIN {X 0,Y 574.103,Z 306.995,A -85,B 0,C 180,E1 -2324.695,E2 -2324.695} C_VEL
LIN {X 0,Y 573.951,Z 321.002,A -85,B 0,C 180,E1 -2325.27,E2 -2325.27} C_VEL
LIN {X 0,Y 573.757,Z 333.152,A -85,B 0,C 180,E1 -2325.91,E2 -2325.91} C_VEL
LIN {X 0,Y 573.631,Z 345.457,A -85,B 0,C 180,E1 -2326.72,E2 -2326.72} C_VEL
LIN {X 0,Y 573.477,Z 356.67,A -85,B 0,C 180,E1 -2327.616,E2 -2327.616} C_VEL
LIN {X 0,Y 573.328,Z 367.649,A -85,B 0,C 180,E1 -2328.689,E2 -2328.689} C_VEL
LIN {X 0,Y 573.231,Z 376.716,A -85,B 0,C 180,E1 -2329.76,E2 -2329.76} C_VEL
LIN {X 0,Y 573.134,Z 385.36,A -85,B 0,C 180,E1 -2331.005,E2 -2331.005} C_VEL
LIN {X 0,Y 573.063,Z 392.33,A -85,B 0,C 180,E1 -2332.247,E2 -2332.247} C_VEL
LIN {X 0,Y 573.031,Z 397.661,A -85,B 0,C 180,E1 -2333.432,E2 -2333.432} C_VEL
LIN {X 0,Y 572.996,Z 402.154,A -85,B 0,C 180,E1 -2334.722,E2 -2334.722} C_VEL
LIN {X 0,Y 573.008,Z 404.899,A -85,B 0,C 180,E1 -2335.78,E2 -2335.78} C_VEL
LIN {X 0,Y 572.955,Z 407.337,A -85,B 0,C 180,E1 -2337.188,E2 -2337.188} C_VEL
LIN {X 0,Y 572.946,Z 408.416,A -85,B 0,C 180,E1 -2338.594,E2 -2338.594} C_VEL
LIN {X 0,Y 572.937,Z 408.174,A -85,B 0,C 180,E1 -2340,E2 -2340} C_VEL
LIN {X 0,Y 572.948,Z 406.637,A -85,B 0,C 180,E1 -2341.406,E2 -2341.406} C_VEL
LIN {X 0,Y 572.963,Z 403.699,A -85,B 0,C 180,E1 -2342.812,E2 -2342.812} C_VEL
LIN {X 0,Y 573.033,Z 399.331,A -85,B 0,C 180,E1 -2344.22,E2 -2344.22} C_VEL
LIN {X 0,Y 573.068,Z 393.379,A -85,B 0,C 180,E1 -2345.631,E2 -2345.631} C_VEL
LIN {X 0,Y 573.075,Z 386.983,A -85,B 0,C 180,E1 -2346.82,E2 -2346.82} C_VEL
LIN {X 0,Y 573.178,Z 378.4,A -85,B 0,C 180,E1 -2348.106,E2 -2348.106} C_VEL
LIN {X 0,Y 573.297,Z 369.765,A -85,B 0,C 180,E1 -2349.17,E2 -2349.17} C_VEL
LIN {X 0,Y 573.436,Z 359.273,A -85,B 0,C 180,E1 -2350.237,E2 -2350.237} C_VEL
LIN {X 0,Y 573.578,Z 348.767,A -85,B 0,C 180,E1 -2351.124,E2 -2351.124} C_VEL
LIN {X 0,Y 573.725,Z 337.388,A -85,B 0,C 180,E1 -2351.921,E2 -2351.921} C_VEL
LIN {X 0,Y 573.898,Z 324.6,A -85,B 0,C 180,E1 -2352.645,E2 -2352.645} C_VEL
LIN {X 0,Y 574.06,Z 311.572,A -85,B 0,C 180,E1 -2353.226,E2 -2353.226} C_VEL
LIN {X 0,Y 574.109,Z 305.439,A -85,B 0,C 180,E1 -2353.45,E2 -2353.45} C_VEL
LIN {X 0,Y 573.353,Z 302.23,A -85,B 0,C 180,E1 -2353.603,E2 -2353.603} C_VEL
LIN {X 0,Y 573.302,Z 301.766,A -85,B 0,C 180,E1 -2353.74,E2 -2353.74} C_VEL
LIN {X 0,Y 573.264,Z 301.704,A -85,B 0,C 180,E1 -2357.01,E2 -2357.01} C_VEL
LIN {X 0,Y 573.272,Z 301.698,A -85,B 0,C 180,E1 -2359.415,E2 -2359.415} C_VEL
LIN {X 0,Y 572.573,Z 301.785,A -85,B 0,C 180,E1 -2360.002,E2 -2360.002} C_VEL
LIN {X 0,Y 569.689,Z 302.149,A -85,B 0,C 180,E1 -2360.954,E2 -2360.954} C_VEL
LIN {X 0,Y 567.277,Z 302.446,A -85,B 0,C 180,E1 -2361.72,E2 -2361.72} C_VEL
LIN {X 0,Y 566.256,Z 302.573,A -85,B 0,C 180,E1 -2362.311,E2 -2362.311} C_VEL
LIN {X 0,Y 566.18,Z 302.585,A -85,B 0,C 180,E1 -2362.512,E2 -2362.512} C_VEL
LIN {X 0,Y 566.223,Z 302.578,A -85,B 0,C 180,E1 -2365.03,E2 -2365.03} C_VEL
LIN {X 0,Y 566.216,Z 302.575,A -85,B 0,C 180,E1 -2367.339,E2 -2367.339} C_VEL
